// Canale 6 - Totale pacchi quinto codice - parziale
Counters[6].Enable := TRUE;
Counters[6].Nome := CONCAT(STR1:= 'Quinto codice - parziale, VALORE -> ', STR2 := INT_TO_STRING(5));
Counters[6].Enable_Reset_Storico := FALSE;
Counters[6].ResetCounter := DATA_LOGGER.Reset_Operatore;
Counters[6].Daily_Reference_Total := Counters[1].Daily_Counter_State;
Counters[6].Weekly_Reference_Total := Counters[1].Weekly_Counter_State;
Counters[6].Periodic_Reference_Total := TotalePacchiParziali;
Counters[6].Enable_Reset_Dopo_Salvataggio := TRUE;

// Canale 7 - Totale pacchi sesto codice - parziale
Counters[7].Enable := TRUE;
Counters[7].Nome := CONCAT(STR1:= 'Sesto codice - parziale, VALORE -> ', STR2 := INT_TO_STRING(6));
Counters[7].Enable_Reset_Storico := FALSE;
Counters[7].ResetCounter := DATA_LOGGER.Reset_Operatore;
Counters[7].Daily_Reference_Total := Counters[1].Daily_Counter_State;
Counters[7].Weekly_Reference_Total := Counters[1].Weekly_Counter_State;
Counters[7].Periodic_Reference_Total := TotalePacchiParziali;
Counters[7].Enable_Reset_Dopo_Salvataggio := TRUE;

// Canale 8 - Totale pacchi settimo codice - parziale
Counters[8].Enable := TRUE;
Counters[8].Nome := CONCAT(STR1:= 'Settimo codice - parziale, VALORE -> ', STR2 := INT_TO_STRING(7));
Counters[8].Enable_Reset_Storico := FALSE;
Counters[8].ResetCounter := DATA_LOGGER.Reset_Operatore;
Counters[8].Daily_Reference_Total := Counters[1].Daily_Counter_State;
Counters[8].Weekly_Reference_Total := Counters[1].Weekly_Counter_State;
Counters[8].Periodic_Reference_Total := TotalePacchiParziali;
Counters[8].Enable_Reset_Dopo_Salvataggio := TRUE;

// Canale 9 - Totale pacchi ottavo codice - parziale
Counters[9].Enable := TRUE;
Counters[9].Nome := CONCAT(STR1:= 'Ottavo codice - parziale, VALORE -> ', STR2 := INT_TO_STRING(8));
Counters[9].Enable_Reset_Storico := FALSE;
Counters[9].ResetCounter := DATA_LOGGER.Reset_Operatore;
Counters[9].Daily_Reference_Total := Counters[1].Daily_Counter_State;
Counters[9].Weekly_Reference_Total := Counters[1].Weekly_Counter_State;
Counters[9].Periodic_Reference_Total := TotalePacchiParziali;
Counters[9].Enable_Reset_Dopo_Salvataggio := TRUE;

// Canale 10 - Totale pacchi nono codice - parziale
Counters[10].Enable := TRUE;
Counters[10].Nome := CONCAT(STR1:= 'Nono codice - parziale, VALORE -> ', STR2 := INT_TO_STRING(9));
Counters[10].Enable_Reset_Storico := FALSE;
Counters[10].ResetCounter := DATA_LOGGER.Reset_Operatore;
Counters[10].Daily_Reference_Total := Counters[1].Daily_Counter_State;
Counters[10].Weekly_Reference_Total := Counters[1].Weekly_Counter_State;
Counters[10].Periodic_Reference_Total := TotalePacchiParziali;
Counters[10].Enable_Reset_Dopo_Salvataggio := TRUE;

// Canale 11 - Totale pacchi decimo codice - parziale
Counters[11].Enable := TRUE;
Counters[11].Nome := CONCAT(STR1:= 'Decimo codice - parziale, VALORE -> ', STR2 := INT_TO_STRING(10));
Counters[11].Enable_Reset_Storico := FALSE;
Counters[11].ResetCounter := DATA_LOGGER.Reset_Operatore;
Counters[11].Daily_Reference_Total := Counters[1].Daily_Counter_State;
Counters[11].Weekly_Reference_Total := Counters[1].Weekly_Counter_State;
Counters[11].Periodic_Reference_Total := TotalePacchiParziali;
Counters[11].Enable_Reset_Dopo_Salvataggio := TRUE;

// Canale 12 - Totale pacchi undicesimo codice - parziale
Counters[12].Enable := TRUE;
Counters[12].Nome := CONCAT(STR1:= 'Undicesimo codice - parziale, VALORE -> ', STR2 := INT_TO_STRING(11));
Counters[12].Enable_Reset_Storico := FALSE;
Counters[12].ResetCounter := DATA_LOGGER.Reset_Operatore;
Counters[12].Daily_Reference_Total := Counters[1].Daily_Counter_State;
Counters[12].Weekly_Reference_Total := Counters[1].Weekly_Counter_State;
Counters[12].Periodic_Reference_Total := TotalePacchiParziali;
Counters[12].Enable_Reset_Dopo_Salvataggio := TRUE;

// Canale 13 - Totale pacchi dodicesimo codice - parziale
Counters[13].Enable := TRUE;
Counters[13].Nome := CONCAT(STR1:= 'Dodicesimo codice - parziale, VALORE -> ', STR2 := INT_TO_STRING(12));
Counters[13].Enable_Reset_Storico := FALSE;
Counters[13].ResetCounter := DATA_LOGGER.Reset_Operatore;
Counters[13].Daily_Reference_Total := Counters[1].Daily_Counter_State;
Counters[13].Weekly_Reference_Total := Counters[1].Weekly_Counter_State;
Counters[13].Periodic_Reference_Total := TotalePacchiParziali;
Counters[13].Enable_Reset_Dopo_Salvataggio := TRUE;

// Canale 14 - Totale pacchi tredicesimo codice - parziale
Counters[14].Enable := TRUE;
Counters[14].Nome := CONCAT(STR1:= 'Tredicesimo codice - parziale, VALORE -> ', STR2 := INT_TO_STRING(13));
Counters[14].Enable_Reset_Storico := FALSE;
Counters[14].ResetCounter := DATA_LOGGER.Reset_Operatore;
Counters[14].Daily_Reference_Total := Counters[1].Daily_Counter_State;
Counters[14].Weekly_Reference_Total := Counters[1].Weekly_Counter_State;
Counters[14].Periodic_Reference_Total := TotalePacchiParziali;
Counters[14].Enable_Reset_Dopo_Salvataggio := TRUE;

// Canale 15 - Totale pacchi quattordicesimo codice - parziale
Counters[15].Enable := TRUE;
Counters[15].Nome := CONCAT(STR1:= 'Quattordicesimo codice - parziale, VALORE -> ', STR2 := INT_TO_STRING(14));
Counters[15].Enable_Reset_Storico := FALSE;
Counters[15].ResetCounter := DATA_LOGGER.Reset_Operatore;
Counters[15].Daily_Reference_Total := Counters[1].Daily_Counter_State;
Counters[15].Weekly_Reference_Total := Counters[1].Weekly_Counter_State;
Counters[15].Periodic_Reference_Total := TotalePacchiParziali;
Counters[15].Enable_Reset_Dopo_Salvataggio := TRUE;

// Canale 16 - Totale pacchi quindicesimo codice - parziale
Counters[16].Enable := TRUE;
Counters[16].Nome := CONCAT(STR1:= 'Quindicesimo codice - parziale, VALORE -> ', STR2 := INT_TO_STRING(15));
Counters[16].Enable_Reset_Storico := FALSE;
Counters[16].ResetCounter := DATA_LOGGER.Reset_Operatore;
Counters[16].Daily_Reference_Total := Counters[1].Daily_Counter_State;
Counters[16].Weekly_Reference_Total := Counters[1].Weekly_Counter_State;
Counters[16].Periodic_Reference_Total := TotalePacchiParziali;
Counters[16].Enable_Reset_Dopo_Salvataggio := TRUE;

(* Reset x evitare false letture *)
PaccoPresoXDataLogger := FALSE;
//DATA_LOGGER.Reset_Operatore := FALSE;
END_ACTION

ACTION _09_CalcolaFormatura:
//Ack 
IF HMI_ErrAckCalcolaFormatura THEN
	HMI_Forming_ErroreCalcoli := 0;
	HMI_ErrAckCalcolaFormatura := FALSE;
	FOR i:= 1 TO MAXFORMING DO
		HMI_Forming_FormaturaAttivata[i] := FALSE;
	END_FOR
END_IF

//Attivazione
FOR i:= 1 TO MAXFORMING DO
	//IF HMI_Forming_Attivazione[i] AND i <=2 AND FALSE THEN
	IF HMI_Forming_Attivazione[i] AND i <=3 AND FALSE THEN
		NCodiciPresenti := 0;
		FOR iform := 1 TO MAXFORMING DO
			FOR icode:=1 TO MAXFORMINGCODE DO
				FOR icode2:=1 TO MAXFORMINGCODE DO
					IF HMI_Forming_CodiciAbilitatiFormatura[i].Code[icode] = Forming[iform].Code[icode] AND Forming[iform].Code[icode] > 0 AND iform <> i THEN
						HMI_Forming_ErroreCalcoli := ErrRipetizioneCodici;		
						HMI_Forming_Attivazione[i] := FALSE; // prueva quitar 
						RETURN;
					END_IF 
				END_FOR
				IF HMI_Forming_CodiciAbilitatiFormatura[i].Code[icode] > 0 THEN
					NCodiciPresenti := NcodiciPresenti+1;
				END_IF
			END_FOR
		END_FOR
		//VErifico che ci sia almento un codice da attivare
		IF NcodiciPresenti = 0 THEN
			HMI_Forming_ErroreCalcoli := ErrNessunCodiciPresente;
			RETURN;
		END_IF
	
		// MEMSET(ADR(Forming[i]),0,SIZEOF(Forming[i])); //prueva Quitar
		IF NOT CalcolaFormaturaTrig AND FALSE  THEN
			HMI_Forming_FormaturaAttivata[i] 	:= FALSE;
			TFCalcoloFormatura.PulisciMemoria 	:= TRUE;
			IF TFCalcoloFormatura.PulisciMemoriaDone THEN	
				HMI_Forming_ErroreCalcoli := 0;
				//Assegno l'ordine tutto a 1 perchè ho solo lastre
				FOR i:= 1 TO MAXFORMINGSLAB DO
					IF i <= HMI_Forming_NumeroElementiDaDepositare THEN
						TFCalcoloFormatura.TipoElementoDep[i] := LASTRA;//Settiamo tutte lastre!!
					ELSE
						TFCalcoloFormatura.TipoElementoDep[i] := TERMINATORE;//Settiamo il resto come terminatore
					END_IF
				END_FOR
				TFCalcoloFormatura.Materiale[e_Tipo_Elemento_Da_Lavorare.LASTRA]		:= HMI_Forming_LastraDaDepositare;
				TFCalcoloFormatura.Materiale[e_Tipo_Elemento_Da_Lavorare.LASTRA].Typology := LASTRA;
				TFCalcoloFormatura.Materiale[e_Tipo_Elemento_Da_Lavorare.FALDA]			:= HMI_Forming_LastraDaDepositare;
				TFCalcoloFormatura.Materiale[e_Tipo_Elemento_Da_Lavorare.FALDA].Typology := FALDA;
				TFCalcoloFormatura.Materiale[e_Tipo_Elemento_Da_Lavorare.QUADROTTA]		:= HMI_Forming_LastraDaDepositare;
				TFCalcoloFormatura.Materiale[e_Tipo_Elemento_Da_Lavorare.QUADROTTA].Typology := QUADROTTA;
				TFCalcoloFormatura.Supporto			:= HMI_Forming_Supporto;	//Assegno la tipologia di supporto
				TFCalcoloFormatura.CalcolaFormatura := TRUE; 		//Lancio esecuzione dei calcoli
				MEMSET(ADR(HMI_Forming_FormaturaCalcolata),0,SIZEOF(HMI_Forming_FormaturaCalcolata));	//Pulisco la memoria di destinazione
				CalcolaFormaturaTrig := TRUE;
				HMI_Forming_Attivazione[i] := FALSE;
				TFCalcoloFormatura.PulisciMemoria := FALSE;
			END_IF
		ELSIF (TFCalcoloFormatura.CalcolaFormaturaDone OR TFCalcoloFormatura.Errore > 0) AND CalcolaFormaturaTrig AND FALSE THEN
			TFCalcoloFormatura.CalcolaFormatura := FALSE;
			IF TFCalcoloFormatura.Errore = 0 THEN
				IDFormatura 			:= IDFormatura+1;
				GUIDFormatura 			:= STRING_TO_UINT(concat(UINT_TO_STRING(NUMERO_MACCHINA),UINT_TO_STRING(IDFormatura)));
				HMI_Forming_GUID 		:= GUIDFormatura;
		
				HMI_Forming_FormaturaCalcolata 	:= TFCalcoloFormatura.FormingSlab;
				MEMSET(ADR(Forming[i]),0,SIZEOF(Forming[i]));	//Pulisco la memoria di destinazione
				Forming[i] 							:= TFCalcoloFormatura.FormingSlab;
				Forming[i].Enable 					:= 1;
				Forming[i].Code 					:= HMI_Forming_CodiciAbilitatiFormatura[i].Code;
				Forming[i].GUID						:= HMI_Forming_GUID;
				Forming[i].Pallet					:= HMI_Forming_Supporto;
				HMI_Forming_IndiceFormaturaAttivata := i;
				HMI_Forming_FormaturaAttivata[i] 	:= TRUE;
			ELSE
				HMI_Forming_ErroreCalcoli := TFCalcoloFormatura.Errore;
			END_IF
			CalcolaFormaturaTrig := FALSE;
			HMI_Forming_Attivazione[i] := FALSE;
		END_IF
	ELSIF HMI_Forming_Attivazione[i] AND FALSE THEN
		memset(destAddr:=ADR(TFCalcoloFormatura.Errore),fillByte:=(UINT_TO_USINT(ErrNumeroMassimoFormatureAmmesse)),n:=SIZEOF(TFCalcoloFormatura.Errore));
	END_IF

	//Disattivazione formatura
	IF HMI_Forming_Disattivazione[i] AND FALSE  THEN
		HMI_Forming_Disattivazione[i] := FALSE;
		MEMSET(ADR(Forming[i]),0,SIZEOF(Forming[i]));	//Pulisco la formatura selezionata e di consegenza la disattivo
	END_IF
		
END_FOR

//IF HMI_Forming_Calcola AND Forming[1].Enable = 1 AND Forming[2].Enable = 1 THEN
//	memset(destAddr:=ADR(TFCalcoloFormatura.Errore),fillByte:=(UINT_TO_USINT(ErrNumeroMassimoFormatureAmmesse)),n:=SIZEOF(TFCalcoloFormatura.Errore));
//	HMI_Forming_Calcola := FALSE;
//Creazione
IF HMI_Forming_Calcola  AND NOT CalcolaFormaturaTrig AND FALSE THEN
	TFCalcoloFormatura.PulisciMemoria := TRUE;
	IF TFCalcoloFormatura.PulisciMemoriaDone THEN	
		HMI_Forming_ErroreCalcoli := 0;
		//Assegno l'ordine tutto a 1 perchè ho solo lastre
		FOR i:= 1 TO MAXFORMINGSLAB DO
			IF i <= HMI_Forming_NumeroElementiDaDepositare THEN
				TFCalcoloFormatura.TipoElementoDep[i] := LASTRA;//Settiamo tutte lastre!!
			ELSE
				TFCalcoloFormatura.TipoElementoDep[i] := TERMINATORE;//Settiamo il resto come terminatore
			END_IF
		END_FOR
		TFCalcoloFormatura.Materiale[e_Tipo_Elemento_Da_Lavorare.LASTRA]		:= HMI_Forming_LastraDaDepositare;
		TFCalcoloFormatura.Materiale[e_Tipo_Elemento_Da_Lavorare.LASTRA].Typology := LASTRA;
		TFCalcoloFormatura.Materiale[e_Tipo_Elemento_Da_Lavorare.FALDA]			:= HMI_Forming_LastraDaDepositare;
		TFCalcoloFormatura.Materiale[e_Tipo_Elemento_Da_Lavorare.FALDA].Typology := FALDA;
		TFCalcoloFormatura.Materiale[e_Tipo_Elemento_Da_Lavorare.QUADROTTA]		:= HMI_Forming_LastraDaDepositare;
		TFCalcoloFormatura.Materiale[e_Tipo_Elemento_Da_Lavorare.QUADROTTA].Typology := QUADROTTA;
		TFCalcoloFormatura.Supporto					:= HMI_Forming_Supporto;	//Assegno la tipologia di supporto
		TFCalcoloFormatura.CalcolaFormatura 		:= HMI_Forming_Calcola; 		//Lancio esecuzione dei calcoli
		TFCalcoloFormatura.NumeroElementiDaDepositare := HMI_Forming_NumeroElementiDaDepositare; 		//Lancio esecuzione dei calcoli
			
		MEMSET(ADR(HMI_Forming_FormaturaCalcolata),0,SIZEOF(HMI_Forming_FormaturaCalcolata));	//Pulisco la memoria di destinazione
		CalcolaFormaturaTrig := TRUE;
		//HMI_Forming_Calcola := FALSE;
		TFCalcoloFormatura.PulisciMemoria := FALSE;
	END_IF

ELSIF HMI_Forming_Calcola AND (TFCalcoloFormatura.CalcolaFormaturaDone OR TFCalcoloFormatura.Errore > 0) AND CalcolaFormaturaTrig AND FALSE THEN
	HMI_Forming_Calcola := FALSE;
	TFCalcoloFormatura.CalcolaFormatura := FALSE;
	IF TFCalcoloFormatura.Errore = 0 THEN
		HMI_Forming_FormaturaCalcolata 	:= TFCalcoloFormatura.FormingSlab;
	//	IDFormatura 			:= IDFormatura+1;
	//	GUIDFormatura 			:= STRING_TO_UINT(concat(UINT_TO_STRING(NUMERO_MACCHINA),UINT_TO_STRING(IDFormatura)));
	//	HMI_Forming_GUID 		:= GUIDFormatura;
		(*FOR i:= 1 TO 2 DO
			IF Forming[i].Enable <> 1 THEN
				MEMSET(ADR(Forming[i]),0,SIZEOF(Forming[i]));	//Pulisco la memoria di destinazione
				HMI_Forming_IndiceFormaturaAttivata := i;
				Forming[i] 			:= TFCalcoloFormatura.FormingSlab;
				Forming[i].Enable 	:= 1;
				Forming[i].Code 	:= HMI_Forming_CodiciAbilitatiFormatura[i].Code;
				Forming[i].GUID		:= HMI_Forming_GUID;
				Forming[i].Pallet	:= HMI_Forming_Supporto;
			ELSE
				CONTINUE;
			END_IF
			EXIT;
		END_FOR*)
		HMI_Forming_FormaturaCreata := TRUE;
	ELSE
		HMI_Forming_ErroreCalcoli := TFCalcoloFormatura.Errore;
	END_IF
	
	CalcolaFormaturaTrig := FALSE;
END_IF
IF FALSE THEN 
	 TFCalcoloFormatura();
END_IF
  

(*//Ack 
IF HMI_ErrAckCalcolaFormatura THEN
	HMI_Forming_ErroreCalcoli := 0;
	HMI_ErrAckCalcolaFormatura := FALSE;
	FOR i:= 1 TO MAXFORMING DO
		HMI_ConfermaAttivazioneFormatura[i] := FALSE;
		HMI_Forming_FormaturaAttivata[i] := FALSE;
	END_FOR
END_IF

//Attivazione
FOR i:= 1 TO MAXFORMING DO
	IF HMI_Forming_Attivazione[i] AND i <=2 THEN
		NCodiciPresenti := 0;
		
		FOR iform := 1 TO MAXFORMING DO
			FOR icode:=1 TO MAXFORMINGCODE DO
				FOR icode2:=1 TO MAXFORMINGCODE DO
					IF HMI_Forming_CodiciAbilitatiFormatura[i].Code[icode] = Forming[iform].Code[icode] AND Forming[iform].Code[icode] > 0 AND iform <> i THEN
						HMI_Forming_ErroreCalcoli := ErrRipetizioneCodici;		
						HMI_Forming_Attivazione[i] := FALSE;
						RETURN;
					END_IF 
				END_FOR
				IF HMI_Forming_CodiciAbilitatiFormatura[i].Code[icode] > 0 THEN
					NCodiciPresenti := NcodiciPresenti+1;
				END_IF
			END_FOR
		END_FOR
		//VErifico che ci sia almento un codice da attivare
		IF NcodiciPresenti = 0 THEN
			HMI_Forming_ErroreCalcoli := ErrNessunCodiciPresente;
			RETURN;
		END_IF
	
		MEMSET(ADR(Forming[i]),0,SIZEOF(Forming[i]));
		IF NOT CalcolaFormaturaTrig  THEN
			HMI_Forming_FormaturaAttivata[i] 	:= FALSE;
			TFCalcoloFormatura.PulisciMemoria 	:= TRUE;
			IF TFCalcoloFormatura.PulisciMemoriaDone THEN	
				HMI_Forming_ErroreCalcoli := 0;
				//Assegno l'ordine tutto a 1 perchè ho solo lastre
				FOR i:= 1 TO MAXFORMINGSLAB DO
					IF i <= HMI_Forming_NumeroElementiDaDepositare THEN
						TFCalcoloFormatura.TipoElementoDep[i] := LASTRA;//Settiamo tutte lastre!!
					ELSE
						TFCalcoloFormatura.TipoElementoDep[i] := TERMINATORE;//Settiamo il resto come terminatore
					END_IF
				END_FOR
				TFCalcoloFormatura.Materiale[e_Tipo_Elemento_Da_Lavorare.LASTRA]		:= HMI_Forming_LastraDaDepositare;
				TFCalcoloFormatura.Materiale[e_Tipo_Elemento_Da_Lavorare.LASTRA].Typology := LASTRA;
				TFCalcoloFormatura.Materiale[e_Tipo_Elemento_Da_Lavorare.FALDA]			:= HMI_Forming_LastraDaDepositare;
				TFCalcoloFormatura.Materiale[e_Tipo_Elemento_Da_Lavorare.FALDA].Typology := FALDA;
				TFCalcoloFormatura.Materiale[e_Tipo_Elemento_Da_Lavorare.QUADROTTA]		:= HMI_Forming_LastraDaDepositare;
				TFCalcoloFormatura.Materiale[e_Tipo_Elemento_Da_Lavorare.QUADROTTA].Typology := QUADROTTA;
				TFCalcoloFormatura.Supporto			:= HMI_Forming_Supporto;	//Assegno la tipologia di supporto
				TFCalcoloFormatura.CalcolaFormatura := TRUE; 		//Lancio esecuzione dei calcoli
				MEMSET(ADR(HMI_Forming_FormaturaCalcolata),0,SIZEOF(HMI_Forming_FormaturaCalcolata));	//Pulisco la memoria di destinazione
				HMI_Forming_Attivazione[i] := FALSE;
				TFCalcoloFormatura.PulisciMemoria := FALSE;
				CalcolaFormaturaTrig := TRUE;
			END_IF
		ELSIF (TFCalcoloFormatura.CalcolaFormaturaDone OR TFCalcoloFormatura.Errore > 0) AND CalcolaFormaturaTrig THEN
			//CalcolaFormaturaTrig := FALSE;
			TFCalcoloFormatura.CalcolaFormatura := FALSE;
			IF TFCalcoloFormatura.Errore = 0 THEN
				IDFormatura 			:= IDFormatura+1;
				GUIDFormatura 			:= STRING_TO_UINT(concat(UINT_TO_STRING(NUMERO_MACCHINA),UINT_TO_STRING(IDFormatura)));
				HMI_Forming_GUID 		:= GUIDFormatura;
		
				HMI_Forming_FormaturaCalcolata 	:= TFCalcoloFormatura.FormingSlab;
				MEMSET(ADR(Forming[i]),0,SIZEOF(Forming[i]));	//Pulisco la memoria di destinazione
				Forming[i] 							:= TFCalcoloFormatura.FormingSlab;
				Forming[i].Enable 					:= 1;
				Forming[i].Code 					:= HMI_Forming_CodiciAbilitatiFormatura[i].Code;
				Forming[i].GUID						:= HMI_Forming_GUID;
				Forming[i].Pallet					:= HMI_Forming_Supporto;
				HMI_Forming_IndiceFormaturaAttivata := i;
				HMI_Forming_FormaturaAttivata[i] 	:= TRUE;
			ELSE
				HMI_Forming_ErroreCalcoli := TFCalcoloFormatura.Errore;
			END_IF
			HMI_Forming_Attivazione[i] := FALSE;
		END_IF
	ELSIF HMI_Forming_Attivazione[i] THEN
		memset(destAddr:=ADR(TFCalcoloFormatura.Errore),fillByte:=(UINT_TO_USINT(ErrNumeroMassimoFormatureAmmesse)),n:=SIZEOF(TFCalcoloFormatura.Errore));
	END_IF

	//Disattivazione formatura
	IF HMI_Forming_Disattivazione[i] THEN
		HMI_Forming_Disattivazione[i] := FALSE;
		MEMSET(ADR(Forming[i]),0,SIZEOF(Forming[i]));	//Pulisco la formatura selezionata e di consegenza la disattivo
	END_IF
		
END_FOR

//IF HMI_Forming_Calcola AND Forming[1].Enable = 1 AND Forming[2].Enable = 1 THEN
//	memset(destAddr:=ADR(TFCalcoloFormatura.Errore),fillByte:=(UINT_TO_USINT(ErrNumeroMassimoFormatureAmmesse)),n:=SIZEOF(TFCalcoloFormatura.Errore));
//	HMI_Forming_Calcola := FALSE;
//Creazione
IF HMI_Forming_Calcola  AND NOT CalcolaFormaturaTrig  THEN
	TFCalcoloFormatura.PulisciMemoria := TRUE;
	IF TFCalcoloFormatura.PulisciMemoriaDone THEN	
		TFCalcoloFormatura.PulisciMemoria := FALSE;
		HMI_Forming_ErroreCalcoli := 0;
		CalcolaFormaturaTrig := TRUE;
		//Assegno l'ordine tutto a 1 perchè ho solo lastre
		FOR i:= 1 TO MAXFORMINGSLAB DO
			IF i <= HMI_Forming_NumeroElementiDaDepositare THEN
				TFCalcoloFormatura.TipoElementoDep[i] := LASTRA;//Settiamo tutte lastre!!
			ELSE
				TFCalcoloFormatura.TipoElementoDep[i] := TERMINATORE;//Settiamo il resto come terminatore
			END_IF
		END_FOR
		TFCalcoloFormatura.Materiale[e_Tipo_Elemento_Da_Lavorare.LASTRA]		:= HMI_Forming_LastraDaDepositare;
		TFCalcoloFormatura.Materiale[e_Tipo_Elemento_Da_Lavorare.LASTRA].Typology := LASTRA;
		TFCalcoloFormatura.Materiale[e_Tipo_Elemento_Da_Lavorare.FALDA]			:= HMI_Forming_LastraDaDepositare;
		TFCalcoloFormatura.Materiale[e_Tipo_Elemento_Da_Lavorare.FALDA].Typology := FALDA;
		TFCalcoloFormatura.Materiale[e_Tipo_Elemento_Da_Lavorare.QUADROTTA]		:= HMI_Forming_LastraDaDepositare;
		TFCalcoloFormatura.Materiale[e_Tipo_Elemento_Da_Lavorare.QUADROTTA].Typology := QUADROTTA;
		TFCalcoloFormatura.Supporto					:= HMI_Forming_Supporto;	//Assegno la tipologia di supporto
		TFCalcoloFormatura.CalcolaFormatura 		:= HMI_Forming_Calcola; 		//Lancio esecuzione dei calcoli
		TFCalcoloFormatura.NumeroElementiDaDepositare := HMI_Forming_NumeroElementiDaDepositare; 		//Lancio esecuzione dei calcoli
			
		MEMSET(ADR(HMI_Forming_FormaturaCalcolata),0,SIZEOF(HMI_Forming_FormaturaCalcolata));	//Pulisco la memoria di destinazione
		//HMI_Forming_Calcola := FALSE;
	END_IF

ELSIF HMI_Forming_Calcola AND (TFCalcoloFormatura.CalcolaFormaturaDone OR TFCalcoloFormatura.Errore > 0) AND CalcolaFormaturaTrig THEN
	HMI_Forming_Calcola := FALSE;
	TFCalcoloFormatura.CalcolaFormatura := FALSE;
	IF TFCalcoloFormatura.Errore = 0 THEN
		HMI_Forming_FormaturaCalcolata 	:= TFCalcoloFormatura.FormingSlab;
	//	IDFormatura 			:= IDFormatura+1;
	//	GUIDFormatura 			:= STRING_TO_UINT(concat(UINT_TO_STRING(NUMERO_MACCHINA),UINT_TO_STRING(IDFormatura)));
	//	HMI_Forming_GUID 		:= GUIDFormatura;
		(*FOR i:= 1 TO 2 DO
			IF Forming[i].Enable <> 1 THEN
				MEMSET(ADR(Forming[i]),0,SIZEOF(Forming[i]));	//Pulisco la memoria di destinazione
				HMI_Forming_IndiceFormaturaAttivata := i;
				Forming[i] 			:= TFCalcoloFormatura.FormingSlab;
				Forming[i].Enable 	:= 1;
				Forming[i].Code 	:= HMI_Forming_CodiciAbilitatiFormatura[i].Code;
				Forming[i].GUID		:= HMI_Forming_GUID;
				Forming[i].Pallet	:= HMI_Forming_Supporto;
			ELSE
				CONTINUE;
			END_IF
			EXIT;
		END_FOR*)
		HMI_Forming_FormaturaCreata := TRUE;
	ELSE
		HMI_Forming_ErroreCalcoli := TFCalcoloFormatura.Errore;
	END_IF
	
	CalcolaFormaturaTrig := FALSE;
END_IF

TFCalcoloFormatura();*)
END_ACTION

ACTION _10_PackModifier:
//Filtro le FTC delle postazioni
FOR i := 1 TO MAXAREAPRESENT DO
	FiltroFTCPalletPerManuale[i].FilterTime_OFF := 3000;
	FiltroFTCPalletPerManuale[i].FilterTime_ON 	:= 3000;
	FiltroFTCPalletPerManuale[i].IN_Signal 		:= I_PHPresenzaPallet[i];
	FiltroFTCPalletPerManuale[i]();
END_FOR

IF MachinePalletizer_TF.CmdExe.Code = CmdNOP THEN
	FOR i:= 1 TO MAXAREAPRESENT DO
		IF HMI_NumeroPezziPresentiPostazione[i] <> WorkAreaState[i].P-1 THEN
			WorkAreaState[i].P := HMI_NumeroPezziPresentiPostazione[i]+1;
		END_IF	
		
		IF HMI_NumeroPezziPresentiCavallete[i].HMI_NumeroPezziPresentiPostazione_A_Cavaleto <> WorkAreaState[i].P_Cava.HMI_NumeroPezziPresentiPostazione_A_Cavaleto -1	THEN 
			WorkAreaState[i].P_Cava.HMI_NumeroPezziPresentiPostazione_A_Cavaleto 
								:= HMI_NumeroPezziPresentiCavallete[i].HMI_NumeroPezziPresentiPostazione_A_Cavaleto +1 ;
		END_IF
		IF HMI_NumeroPezziPresentiCavallete[i].HMI_NumeroPezziPresentiPostazione_B_Cavaleto <> WorkAreaState[i].P_Cava.HMI_NumeroPezziPresentiPostazione_B_Cavaleto -1	THEN 
			WorkAreaState[i].P_Cava.HMI_NumeroPezziPresentiPostazione_B_Cavaleto 
								:= HMI_NumeroPezziPresentiCavallete[i].HMI_NumeroPezziPresentiPostazione_B_Cavaleto +1 ;
		END_IF
		IF (ActualPickingListFromHMI[1].State <> 0 OR ActualPickingListFromHMI[2].State <> 0 OR ActualPickingListFromHMI[3].State <>0)
				AND WorkAreaState[i].Supporto.Tipologia = CAVALLETTO THEN 
			WorkAreaState[i].P := HMI_NumeroPezziPresentiCavallete[i].HMI_NumeroPezziPresentiPostazione_A_Cavaleto 
					+ HMI_NumeroPezziPresentiCavallete[i].HMI_NumeroPezziPresentiPostazione_B_Cavaleto +1 ;
		END_IF		
		
		IF WorkAreaState[i].PackPointerModified THEN//Se sto facendo una modifica da HMI
			WorkAreaState[i].PackPointer:= MIN(MAX(1,WorkAreaState[i].PackPointer ),MAXFORMINGSLAB);//limito i valori con quelli ammissibili
			IF WorkAreaState[i].PackPointer > WorkAreaState[i].P THEN 
				IF (WorkAreaState[i].PackPointer - WorkAreaState[i].P) = 1 THEN
					WorkAreaState[i].P := WorkAreaState[i].P+1;
				ELSE 
					WorkAreaState[i].P := WorkAreaState[i].PackPointer+1;	
				END_IF
			ELSE
				IF (WorkAreaState[i].PackPointer - WorkAreaState[i].P) = -1 THEN
					WorkAreaState[i].P := WorkAreaState[i].P-1;
				ELSE 
					WorkAreaState[i].P := WorkAreaState[i].PackPointer+1;	
				END_IF
			END_IF
			WorkAreaState[i].Slow := 1;
			WorkAreaState[i].PackPointerModified := FALSE;
			WorkAreaState[i].PackPointer := -1;
		END_IF
		//
		HMI_NumeroPezziPresentiPostazione[i] := MAX(0,WorkAreaState[i].P-1);
		
		AggiuntaPalletManuale(WorkArea := ADR(WorkArea),
									WorkAreaState := ADR(WorkAreaState),
									WorkAreaNumber := i,
									Forming := ADR(Forming),
									Pallet := ADR(Pallet),
									Layer := ADR(Layer),
									ProgressiveNrWA := ADR(ProgressiveNrWA),
									CodicePostazione := WorkAreaState[i].Code,
									AbilitaAssegnazioneCodicePiazzoleConPaccoSuRibaltino := TRUE,
									PH_Presenza := FiltroFTCPalletPerManuale[i].Out_Signal_Filtrato);	
	END_FOR
END_IF
END_ACTION

ACTION _11_CalcolaListaProduzione:
{region "Gestione zona GLOBALE - Postazioni da 1 a 8"}


//#############################################################################################################

{region "Gestione zona GLOBALE - Postazioni da 1 a 8"}

//Traferisco i valori dei supporti della lista 1 nella lista 2 e 3
 

FOR LoopLista := 1 TO 3 DO
	IdxLista := LoopLista;		 
	 // IdxLista := 2;		  
	CASE IdxLista OF	 
		1: Iforstart := 1; Iforend := MAXAREAPRESENT;
		2: Iforstart := 1; Iforend := 4;
		3: Iforstart := 5; Iforend := MAXAREAPRESENT;
	END_CASE	 
	IF MachinePalletizer_TF.IN.Mode.Man AND
		(MachinePalletizer_TF.CmdExe.Code = CmdNOP OR MachinePalletizer_TF.CmdExe.Code = CmdMAN) THEN

//--------------------------------------------------------
			//AZZERAMENTO (Reset) lista di picking	
//--------------------------------------------------------		 
			IF Cmd_AzzeraLista[IdxLista] THEN
				IF Prueva THEN
					MissionClr := ADR(Mission) ;
	 				MEMSET(destAddr := ADR(MissionClr^),fillByte := 0 , n := SIZEOF(MissionClr^));
				END_IF
					ClrEstructura := ADR(PosCavalleteOrdenPikin) ;
					MEMSET(destAddr := ADR(ClrEstructura^),fillByte := 0 , n := SIZEOF(ClrEstructura^));	  
					NuEstacionesPiking := 0 ;	  
					NuEstacionPiking   := 0 ;
					NuPosGuiroPiking := 0;
					PosFinOrdenPikingCaballete := 0 ;
					
					MultiplesCavalletesReceta := FALSE ;
					CoordenadaPasillo0_Y := 0 ;
					CoordenadaPasillo180_Y := 0 ;
				
				//FOR i:= 1 TO 3 DO
						//CalcolaFormingRT2[i] := FALSE ;
					CalcolaFormingRT[IdxLista] := FALSE ;
					CalcolaFormingRT2[IdxLista] := FALSE ;	 
						//#Añadido 4_7_2025########################
					Formacion_bandelCalOk[IdxLista]			:= FALSE ;
					Formacion_FrameCalOk[IdxLista]			:= FALSE ;
					Formacion_De_listaOk[IdxLista]			:= FALSE ;
					FormaturaAFRAMERT[IdxLista]		   	:=	FormingEmpty;
					FormaturaBundleRT[IdxLista]	 		:=	FormingEmpty;
					
					MEMSET(destAddr := ADR(TFFormacionBandelCalculada),fillByte := 0 , n := SIZEOF(TFFormacionBandelCalculada));
					MEMSET(destAddr := ADR(TFFormacionCavalleteCalculada),fillByte := 0 , n := SIZEOF(TFFormacionCavalleteCalculada));
					MEMSET(destAddr := ADR(TFCalcoloFormaturaWA),fillByte := 0 , n := SIZEOF(TFCalcoloFormaturaWA));
					MEMSET(destAddr := ADR(GestionCargaCaballete),fillByte := 0 , n := SIZEOF(GestionCargaCaballete));	
					MEMSET(destAddr := ADR(GestionDescargaCaballete),fillByte := 0 , n := SIZEOF(GestionDescargaCaballete));			  
				//Añadido 4_7_2025##########################
						
				// END_FOR
				ActualPickingListFromHMI[IdxLista].State := e_StatoWorkOrder.NON_ESEGUITO;
				HMI_NumeroLastreDepOrdineAttuale[IdxLista] := 0; 
				//Disattivazione formatura
				Forming[1] := FormingEmpty;	//Pulisco la formatura selezionata e di consegenza la disattivo
				Forming[2] := FormingEmpty;	//Pulisco la formatura selezionata e di consegenza la disattivo
				Forming[3] := FormingEmpty;	//Pulisco la formatura selezionata e di consegenza la disattivo
				Forming[4] := FormingEmpty;	//Pulisco la formatura selezionata e di consegenza la disattivo
				ActualPickingListFromHMI[IdxLista].State := e_StatoWorkOrder.NON_ESEGUITO;
				Cmd_AttivaLista[IdxLista] := FALSE;
				HMI_Forming_NumeroElementiDaDepositare := 0;
 				RequestPickingListFromHMI[IdxLista].SlabNumber :=0;
	 
				//Azzero le liste per le postazioni dove non avviene la pallettizzazione
				FOR i:= Iforstart TO Iforend DO	
					TFClearWorkAreaArray(ADR(Workarea),ADR(WorkAreaState),k:=i);
					HMI_WorkAreaDataPicking[i].Destinazione := FALSE;
					HMI_WorkAreaDataPicking[i].NumElementiDaLavorare := 0;
					WorkAreaState[i].P 			:= 1;
					WorkAreaProductionList[i] 	:= ListaEmpty;
					WorkAreaOffset[i].Y 		:= 0;
					//HMI_NumeroPezziPresentiPostazione[i] 	:= 0; // Quitado Para No resetear posiciones
					NumeroPezziPresentiPostazioneStart[i] 	:= 0;
					WorkAreaProductionList[i].Stato 		:= e_Stato_ListaDiProduzione.LISTA_PROD_ASSENTE;	 
				END_FOR			  
				ActualPickingListFromHMI[IdxLista].SlabNumber 		  			:= 0;
				ActualPickingListFromHMI[IdxLista].SlabDimension.XDim 			:= 0;
				ActualPickingListFromHMI[IdxLista].SlabDimension.YDim 			:= 0;
				ActualPickingListFromHMI[IdxLista].SlabDimension.ZDim 			:= 0;
				ActualPickingListFromHMI[IdxLista].SupportPianoLegno 			:= SupportDataEmpty;
				ActualPickingListFromHMI[IdxLista].SupportPianoFerro 			:= SupportDataEmpty;
				ActualPickingListFromHMI[IdxLista].SupportVertBundle 			:= SupportDataEmpty;
				ActualPickingListFromHMI[IdxLista].SupportVertCav 			 	:= SupportDataEmpty;
				
				HMI_ErroreCalcoloLista 		:= 0;
				Cmd_CalcolaLista[IdxLista] 	:= FALSE;
				HMI_Forming_Attivazione[IdxLista] 	:= FALSE;//attivo nuova formatura
				Cmd_AzzeraLista[IdxLista] := FALSE;
				//Ack 
				//IF HMI_ErrAckCalcolaFormatura THEN
					HMI_Forming_ErroreCalcoli := 0;
					HMI_ErrAckCalcolaFormatura := FALSE;
					FOR i:= 1 TO MAXFORMING DO
						HMI_ConfermaAttivazioneFormatura[i] := FALSE;
						HMI_Forming_FormaturaAttivata[i] := FALSE;
					END_FOR
				//END_IF
				CalcolaFormaturaTrig := FALSE;
			END_IF



//--------------------------------------------------------
		// COMANDO ATTIVAZIONE  lista di picking	
//--------------------------------------------------------		 		  
			//Se non ho una Destinazione impostata, Num.pezzi impostato, o Num.pezzi richiesto...
			//	Resetto il comando		
					IF Cmd_AttivaLista[1] = TRUE  THEN
						FOR uu := Iforstart TO Iforend DO
							 	IF	HMI_WorkAreaDataPicking[uu].Typology = CAVALLETTO THEN 
									CASE HMI_WorkAreaDataPicking[uu].TipoTrabajoLado_Cavallete OF 
	 									0:
											HMI_NumeroPezziPresentiPostazione[uu] := HMI_NumeroPezziPresentiCavallete[uu].HMI_NumeroPezziPresentiPostazione_A_Cavaleto +
												 HMI_NumeroPezziPresentiCavallete[uu].HMI_NumeroPezziPresentiPostazione_B_Cavaleto ;
										1:
											HMI_NumeroPezziPresentiPostazione[uu] := HMI_NumeroPezziPresentiCavallete[uu].HMI_NumeroPezziPresentiPostazione_A_Cavaleto ;									 ;
											 
										2:	
		   									HMI_NumeroPezziPresentiPostazione[uu] := HMI_NumeroPezziPresentiCavallete[uu].HMI_NumeroPezziPresentiPostazione_B_Cavaleto ;
												 
									END_CASE
								END_IF 	 
							END_FOR		  
											
													  
																
						IF 	(HMI_WorkAreaDataPicking[1].Destinazione =0 AND 
							HMI_WorkAreaDataPicking[2].Destinazione =0 AND
							HMI_WorkAreaDataPicking[3].Destinazione =0 AND 
							HMI_WorkAreaDataPicking[4].Destinazione =0 AND	 
							HMI_WorkAreaDataPicking[5].Destinazione =0 AND 
							HMI_WorkAreaDataPicking[6].Destinazione =0 AND
							HMI_WorkAreaDataPicking[7].Destinazione =0 AND 
							HMI_WorkAreaDataPicking[8].Destinazione =0)							 
							OR
							(HMI_NumeroPezziPresentiPostazione[1] =0 AND 
							HMI_NumeroPezziPresentiPostazione[2] =0 AND
							HMI_NumeroPezziPresentiPostazione[3] =0 AND 
							HMI_NumeroPezziPresentiPostazione[4] =0 AND
							HMI_NumeroPezziPresentiPostazione[5] =0 AND 
	 						HMI_NumeroPezziPresentiPostazione[6] =0 AND
							HMI_NumeroPezziPresentiPostazione[7] =0 AND 
							HMI_NumeroPezziPresentiPostazione[8] =0)
							OR	 	 
							RequestPickingListFromHMI[1].SlabNumber = 0	 
						THEN
							Cmd_AttivaLista[1] := FALSE;
						 END_IF
					END_IF		  
					IF Cmd_AttivaLista[2] = TRUE  THEN
						FOR uu := Iforstart TO Iforend DO
							 	IF	HMI_WorkAreaDataPicking[uu].Typology = CAVALLETTO THEN 
									CASE HMI_WorkAreaDataPicking[uu].TipoTrabajoLado_Cavallete OF 
	 									0:
											HMI_NumeroPezziPresentiPostazione[uu] := HMI_NumeroPezziPresentiCavallete[uu].HMI_NumeroPezziPresentiPostazione_A_Cavaleto +
												 HMI_NumeroPezziPresentiCavallete[uu].HMI_NumeroPezziPresentiPostazione_B_Cavaleto ;
										1:
											HMI_NumeroPezziPresentiPostazione[uu] := HMI_NumeroPezziPresentiCavallete[uu].HMI_NumeroPezziPresentiPostazione_A_Cavaleto ;									 ;
											 
										2:	
		   									HMI_NumeroPezziPresentiPostazione[uu] := HMI_NumeroPezziPresentiCavallete[uu].HMI_NumeroPezziPresentiPostazione_B_Cavaleto ;
												 
									END_CASE
								END_IF 	 
							END_FOR		  
						IF 	(HMI_WorkAreaDataPicking[1].Destinazione =0 AND 
							HMI_WorkAreaDataPicking[2].Destinazione =0 AND
							HMI_WorkAreaDataPicking[3].Destinazione =0 AND 
							HMI_WorkAreaDataPicking[4].Destinazione =0)
							OR
							(HMI_NumeroPezziPresentiPostazione[1] =0 AND 
							HMI_NumeroPezziPresentiPostazione[2] =0 AND
							HMI_NumeroPezziPresentiPostazione[3] =0 AND 
							HMI_NumeroPezziPresentiPostazione[4] =0)
							OR	 
							RequestPickingListFromHMI[2].SlabNumber = 0	 	 
						THEN
							Cmd_AttivaLista[2] := FALSE;
						 END_IF
					END_IF		
					IF Cmd_AttivaLista[3] = TRUE  THEN
					  FOR uu := Iforstart TO Iforend DO
							 	IF	HMI_WorkAreaDataPicking[uu].Typology = CAVALLETTO THEN 
									CASE HMI_WorkAreaDataPicking[uu].TipoTrabajoLado_Cavallete OF 
	 									0:
											HMI_NumeroPezziPresentiPostazione[uu] := HMI_NumeroPezziPresentiCavallete[uu].HMI_NumeroPezziPresentiPostazione_A_Cavaleto +
												 HMI_NumeroPezziPresentiCavallete[uu].HMI_NumeroPezziPresentiPostazione_B_Cavaleto ;
										1:
											HMI_NumeroPezziPresentiPostazione[uu] := HMI_NumeroPezziPresentiCavallete[uu].HMI_NumeroPezziPresentiPostazione_A_Cavaleto ;									 ;
											 
										2:	
		   									HMI_NumeroPezziPresentiPostazione[uu] := HMI_NumeroPezziPresentiCavallete[uu].HMI_NumeroPezziPresentiPostazione_B_Cavaleto ;
												 
									END_CASE
								END_IF 	 
							END_FOR		  
						IF 	(HMI_WorkAreaDataPicking[5].Destinazione =0 AND 
							HMI_WorkAreaDataPicking[6].Destinazione =0 AND
							HMI_WorkAreaDataPicking[7].Destinazione =0 AND 
							HMI_WorkAreaDataPicking[8].Destinazione =0)
							OR
							(HMI_NumeroPezziPresentiPostazione[5] =0 AND 
							HMI_NumeroPezziPresentiPostazione[6] =0 AND
							HMI_NumeroPezziPresentiPostazione[7] =0 AND 
							HMI_NumeroPezziPresentiPostazione[8] =0)
							OR	 	 
							RequestPickingListFromHMI[3].SlabNumber = 0	 	 
						THEN
							Cmd_AttivaLista[3] := FALSE;
						 END_IF
					END_IF		
{Region "Prmer Bucle cuenta las piezas a coger y rellena el workareastate Con el Tipo Palet"}

			// COMANDO ATTIVAZIONE  lista di picking	
		    IF Cmd_AttivaLista[IdxLista] AND ActualPickingListFromHMI[IdxLista].State <> e_StatoWorkOrder.IN_ESECUZIONE THEN
				ElementiDaDepositare[IdxLista]   :=0;
				HMI_ErroreCalcoloLista := 0;
				HMI_NumeroLastreDepOrdineAttuale[IdxLista] := 0;
				FOR i:= Iforstart TO Iforend DO	
					//HMI_WorkAreaDataPicking[i].Destinazione := FALSE;
					//HMI_WorkAreaDataPicking[i].NumElementiDaLavorare := 0;
					WorkAreaState[i].P := 1;
					WorkAreaProductionList[i] := ListaEmpty;
				END_FOR	 
				
				FOR i:= Iforstart TO Iforend DO	
					IF NOT HMI_WorkAreaDataPicking[i].Destinazione THEN
						ElementiDaDepositare[IdxLista] := ElementiDaDepositare[IdxLista] +HMI_WorkAreaDataPicking[i].NumElementiDaLavorare;
						WorkAreaState[i].P := HMI_WorkAreaDataPicking[i].NumElementiDaLavorare +1;
									   
						CASE HMI_WorkAreaDataPicking[i].Typology OF
							LEGNO_PIANO,TELAIO_PIANO:
								WorkareaState[i].Supporto.Tipologia := e_Tipo_Pallet.CASSA_STANDARD;
							A_FRAME_VERT:	
								WorkareaState[i].Supporto.Tipologia := e_Tipo_Pallet.CAVALLETTO;
								
							IF HMI_WorkAreaDataPicking[i].NumElementiDaLavorare > 0 THEN 
								NuEstacionesPiking := NuEstacionesPiking + 1 ;	
								PosCavalleteOrdenPikin[i]	:=  e_Tipo_Pallet.CAVALLETTO;  
							END_IF
							BUNDLE_VERT:
								WorkareaState[i].Supporto.Tipologia := e_Tipo_Pallet.BUNDLE;	
							
						 ELSE
								WorkareaState[i].Supporto.Tipologia := e_Tipo_Pallet.CASSA_STANDARD;		   
						 END_CASE
					ELSE
						NumPostazioneDeposito := i; NuEstacionPiking := i;
						
						HMI_WorkAreaDataPicking[NumPostazioneDeposito].NumElementiDaLavorare := RequestPickingListFromHMI[IdxLista].SlabNumber;
						CASE HMI_WorkAreaDataPicking[i].Typology OF
							LEGNO_PIANO,TELAIO_PIANO:
								WorkareaState[i].Supporto.Tipologia := e_Tipo_Pallet.CASSA_STANDARD;
							A_FRAME_VERT:	
								WorkareaState[i].Supporto.Tipologia := e_Tipo_Pallet.CAVALLETTO;
								NuEstacionesPiking := NuEstacionesPiking + 1 ;	
								PosCavalleteOrdenPikin[i]	:=  e_Tipo_Pallet.CAVALLETTO;  	 
							BUNDLE_VERT:
								WorkareaState[i].Supporto.Tipologia := e_Tipo_Pallet.BUNDLE;	
								
							
						 ELSE
								WorkareaState[i].Supporto.Tipologia := e_Tipo_Pallet.CASSA_STANDARD;		   
						 END_CASE
					END_IF

		  
//HMI_NumeroPezziPresentiPostazione[i] := WorkAreaState[i].P -1; //NB:cancellato xckè alla attivazione azzerava il num.pezzi presenti sulle postazioni di prelievo
				END_FOR
	
				IF ElementiDaDepositare[IdxLista] <= HMI_WorkAreaDataPicking[NumPostazioneDeposito].NumElementiDaLavorare THEN
					ActualPickingListFromHMI[IdxLista] 				:= RequestPickingListFromHMI[IdxLista];
					ActualPickingListFromHMI[IdxLista].State 		:= e_StatoWorkOrder.DA_ESEGUIRE;

				ELSE
					HMI_ErroreCalcoloLista := 1;
				END_IF
				Cmd_AttivaLista[IdxLista] 				:= FALSE;
				 
			ELSE
				Cmd_AttivaLista[IdxLista] 				:= FALSE;
				 
			END_IF
{endregion}	

{region "Cotas posicione de trabajo"}

//--------------------------------------------------------------------				
//////// attivazione lista di picking : StatoWorkOrder.DA_ESEGUIRE ///
//--------------------------------------------------------------------				
			IF ActualPickingListFromHMI[IdxLista].State = e_StatoWorkOrder.DA_ESEGUIRE  THEN
				ListaInEsecuzione[IdxLista] := FALSE;
				NumeroListaInEsecuzione := 0;
			
				(* Inserimento sequenza di prelievo dalle postazioni in base al quello che l'operatore ha editato da HMI*)
				ElementiDaDepositare[IdxLista] := 0;
				ElementiElaborati[IdxLista]    := 1;
				NumPostazioneDeposito := 0;
				//FOR i:= 1 TO MAXAREAPRESENT DO
				//	WorkAreaState[i].P := 1;
				//END_FOR		
				
				FOR i:= Iforstart TO Iforend DO//---------- For 1 HMI_WorkAreaDataPicking[i].Destinazione 
					IF HMI_WorkAreaDataPicking[i].Destinazione THEN  //-------> Palet destino
						NumPostazioneDeposito := i;
						HMI_WorkAreaDataPicking[NumPostazioneDeposito].NumElementiDaLavorare 	:= RequestPickingListFromHMI[IdxLista].SlabNumber;
						(*CASE HMI_WorkAreaDataPicking[i].Typology OF     // case Pricipal1*)		 
						CASE HMI_WorkAreaDataPicking[NumPostazioneDeposito].Typology OF     // case Pricipal1	
							(* Se ho un legno in piano *)	 
							LEGNO_PIANO:	
								WorkAreaState[NumPostazioneDeposito].Supporto.Code 						:= ActualPickingListFromHMI[IdxLista].SupportPianoLegno.Code;
								WorkAreaState[NumPostazioneDeposito].Supporto.AltezzaDenteRitenuta 		:= ActualPickingListFromHMI[IdxLista].SupportPianoLegno.DimBaseUtile;
								WorkAreaState[NumPostazioneDeposito].Supporto.DimVertice 				:= ActualPickingListFromHMI[IdxLista].SupportPianoLegno.DimVertice;
								WorkAreaState[NumPostazioneDeposito].Supporto.HMAX 						:= ActualPickingListFromHMI[IdxLista].SupportPianoLegno.HMAX;
								WorkAreaState[NumPostazioneDeposito].Supporto.Tipologia 				:= e_Tipo_Pallet.CASSA_STANDARD;//ActualPickingListFromHMI.Support.Tipologia;
								WorkAreaState[NumPostazioneDeposito].Supporto.XDim 						:= ActualPickingListFromHMI[IdxLista].SupportPianoLegno.XDim;
								WorkAreaState[NumPostazioneDeposito].Supporto.YDim 						:= ActualPickingListFromHMI[IdxLista].SupportPianoLegno.YDim;
								WorkAreaState[NumPostazioneDeposito].Supporto.ZDim 						:= ActualPickingListFromHMI[IdxLista].SupportPianoLegno.ZDim;
								WorkAreaOffset[NumPostazioneDeposito].Y 								:= OFFSET_POSTAZIONE_LEGNO + ActualPickingListFromHMI[IdxLista].SupportPianoLegno.YDim/2;//ATTENZIONE!!! per poter lavorare in centro con i supporti pari, questa misura è la distanza tra il riscontro bundle verticale e il centro postazione PARI
								
								CASE HMI_WorkAreaDataPicking[NumPostazioneDeposito].Typology OF
									LEGNO_PIANO:
										 		WorkAreaProductionList[NumPostazioneDeposito].Support := WorkAreaState[NumPostazioneDeposito].Supporto;
												WorkAreaProductionList[NumPostazioneDeposito].Support.Tipologia	:= e_Tipo_Pallet.CASSA_STANDARD; 
									TELAIO_PIANO:
										 		WorkAreaProductionList[NumPostazioneDeposito].Support := WorkAreaState[NumPostazioneDeposito].Supporto;
												WorkAreaProductionList[NumPostazioneDeposito].Support.Tipologia	:= e_Tipo_Pallet.CASSA_STANDARD; 
									BUNDLE_VERT:
										 		WorkAreaProductionList[NumPostazioneDeposito].Support := WorkAreaState[NumPostazioneDeposito].Supporto;
												WorkAreaProductionList[NumPostazioneDeposito].Support.Tipologia	:= e_Tipo_Pallet.BUNDLE; 
												
									A_FRAME_VERT:
										 		WorkAreaProductionList[NumPostazioneDeposito].Support := WorkAreaState[NumPostazioneDeposito].Supporto;
												WorkAreaProductionList[NumPostazioneDeposito].Support.Tipologia	:= e_Tipo_Pallet.CAVALLETTO; 
												
								END_CASE
								FOR j:= Iforstart TO Iforend DO
									IF NOT HMI_WorkAreaDataPicking[j].Destinazione THEN
										IF HMI_WorkAreaDataPicking[j].NumElementiDaLavorare >= 1 THEN
											ElementiDaDepositare[IdxLista] := ElementiElaborati[IdxLista] + HMI_WorkAreaDataPicking[j].NumElementiDaLavorare;
											FOR k := ElementiElaborati[IdxLista] TO ElementiDaDepositare[IdxLista]-1 DO	
												WorkAreaProductionList[NumPostazioneDeposito].PElementList[k].WA_PRELIEVO := j;
												WorkAreaProductionList[NumPostazioneDeposito].PElementList[k].WA_DEPOSITO := i;	
												ElementiElaborati[IdxLista] := ElementiElaborati[IdxLista]+1; 
											END_FOR
											CASE HMI_WorkAreaDataPicking[j].Typology OF 
												(* Se ho una cassa pianale in legno *)
												LEGNO_PIANO:
													WorkAreaState[j].Supporto.Code 					:= ActualPickingListFromHMI[IdxLista].SupportPianoLegno.Code;
													WorkAreaState[j].Supporto.DimBaseUtile		 	:= ActualPickingListFromHMI[IdxLista].SupportPianoLegno.DimBaseUtile;
													WorkAreaState[j].Supporto.AltezzaDenteRitenuta 	:= ActualPickingListFromHMI[IdxLista].SupportPianoLegno.ZDim+20;
													WorkAreaState[j].Supporto.DimVertice 			:= ActualPickingListFromHMI[IdxLista].SupportPianoLegno.DimVertice;
													WorkAreaState[j].Supporto.HMAX 					:= ActualPickingListFromHMI[IdxLista].SupportPianoLegno.HMAX;
													WorkAreaState[j].Supporto.Tipologia 			:= e_Tipo_Pallet.CASSA_STANDARD;//ActualPickingListFromHMI[1].Support.Tipologia;
													WorkAreaState[j].Supporto.XDim 					:= ActualPickingListFromHMI[IdxLista].SupportPianoLegno.XDim;
													WorkAreaState[j].Supporto.YDim 					:= ActualPickingListFromHMI[IdxLista].SupportPianoLegno.YDim;
													WorkAreaState[j].Supporto.ZDim 					:= ActualPickingListFromHMI[IdxLista].SupportPianoLegno.ZDim;
													WorkAreaOffset[j].Y 							:= OFFSET_POSTAZIONE_LEGNO + ActualPickingListFromHMI[IdxLista].SupportPianoLegno.YDim/2;//ATTENZIONE!!! per poter lavorare in centro con i supporti pari, questa misura è la distanza tra il riscontro bundle verticale e il centro postazione PARI
												(* Se ho una cassa pianale in ferro su supporto *)
												TELAIO_PIANO:
													WorkAreaState[j].Supporto.Code 					:= ActualPickingListFromHMI[IdxLista].SupportPianoFerro.Code;
													WorkAreaState[j].Supporto.DimBaseUtile		 	:= ActualPickingListFromHMI[IdxLista].SupportPianoFerro.DimBaseUtile;
													WorkAreaState[j].Supporto.AltezzaDenteRitenuta 	:= ActualPickingListFromHMI[IdxLista].SupportPianoFerro.ZDim+20;
													WorkAreaState[j].Supporto.DimVertice 			:= ActualPickingListFromHMI[IdxLista].SupportPianoFerro.DimVertice;
													WorkAreaState[j].Supporto.HMAX 					:= ActualPickingListFromHMI[IdxLista].SupportPianoFerro.HMAX;
													WorkAreaState[j].Supporto.Tipologia 			:=  e_Tipo_Pallet.CASSA_STANDARD;//ActualPickingListFromHMI[1].Support.Tipologia;
													WorkAreaState[j].Supporto.XDim 					:= ActualPickingListFromHMI[IdxLista].SupportPianoFerro.XDim;
													WorkAreaState[j].Supporto.YDim 					:= ActualPickingListFromHMI[IdxLista].SupportPianoFerro.YDim;
													WorkAreaState[j].Supporto.ZDim 					:= ActualPickingListFromHMI[IdxLista].SupportPianoFerro.ZDim;
													WorkAreaOffset[j].Y 							:= OFFSET_POSTAZIONE_TELAIO - ActualPickingListFromHMI[IdxLista].SupportPianoFerro.YDim/2;//ATTENZIONE!!! per poter lavorare in centro con i supporti pari, questa misura è la distanza tra il riscontro bundle verticale e il centro postazione PARI
												(* Se ho un bundle *)
												BUNDLE_VERT:
													//WorkAreaState[j].P := ElementiDaDepositare;
													WorkAreaState[j].Supporto.Code 					:= ActualPickingListFromHMI[IdxLista].SupportVertBundle.Code;
													WorkAreaState[j].Supporto.DimBaseUtile		 	:= ActualPickingListFromHMI[IdxLista].SupportVertBundle.DimBaseUtile;
													WorkAreaState[j].Supporto.AltezzaDenteRitenuta 	:= ActualPickingListFromHMI[IdxLista].SupportVertBundle.ZDim+20;
													WorkAreaState[j].Supporto.DimVertice 			:= ActualPickingListFromHMI[IdxLista].SupportVertBundle.DimVertice;
													WorkAreaState[j].Supporto.HMAX 					:= ActualPickingListFromHMI[IdxLista].SupportVertBundle.HMAX;
													WorkAreaState[j].Supporto.Tipologia 			:= e_Tipo_Pallet.BUNDLE;//ActualPickingListFromHMI.SupportVert.Tipologia;
													WorkAreaState[j].Supporto.XDim 					:= ActualPickingListFromHMI[IdxLista].SupportVertBundle.XDim;
													WorkAreaState[j].Supporto.YDim 					:= ActualPickingListFromHMI[IdxLista].SupportVertBundle.YDim;
													WorkAreaState[j].Supporto.ZDim 					:= ActualPickingListFromHMI[IdxLista].SupportVertBundle.ZDim;
													WorkAreaState[j].Supporto.ZDim_Ext1        		:= WorkAreaState[j].Supporto.ZDim + 20;
													//Lo que HABIA	
													//WorkAreaOffset[j].Y 							:= HMI_OffsetDepositoLastra.Y180 ;
													//Mod 25/&/2025	  
													WorkAreaOffset[NumPostazioneDeposito].Y 		:= ActualPickingListFromHMI[IdxLista].SupportVertBundle.YDim-ActualPickingListFromHMI[IdxLista].SupportVertBundle.DimBaseUtile -40 ;			
												(* Se ho un A_Frame *)	  
												A_FRAME_VERT:  						
													//WorkAreaState[j].P := ElementiDaDepositare;
													WorkAreaState[j].Supporto.Code 					:= ActualPickingListFromHMI[IdxLista].SupportVertCav.Code;
													WorkAreaState[j].Supporto.DimBaseUtile		 	:= ActualPickingListFromHMI[IdxLista].SupportVertCav.DimBaseUtile;
													WorkAreaState[j].Supporto.AltezzaDenteRitenuta 	:= ActualPickingListFromHMI[IdxLista].SupportVertCav.ZDim+20;
													WorkAreaState[j].Supporto.DimVertice 			:= ActualPickingListFromHMI[IdxLista].SupportVertCav.DimVertice;
													WorkAreaState[j].Supporto.HMAX 					:= ActualPickingListFromHMI[IdxLista].SupportVertCav.HMAX;
													WorkAreaState[j].Supporto.Tipologia 			:= CAVALLETTO;//ActualPickingListFromHMI.SupportVertCav.Tipologia;
													WorkAreaState[j].Supporto.XDim 					:= ActualPickingListFromHMI[IdxLista].SupportVertCav.XDim;
													WorkAreaState[j].Supporto.YDim 					:= ActualPickingListFromHMI[IdxLista].SupportVertCav.YDim;
													WorkAreaState[j].Supporto.ZDim 					:= ActualPickingListFromHMI[IdxLista].SupportVertCav.ZDim;
													WorkAreaState[j].Supporto.ZDim_Ext1        		:= WorkAreaState[j].Supporto.ZDim + 20;	
													WorkAreaState[j].Supporto.TipoTrabajoLado_Cavallete := HMI_WorkAreaDataPicking[j].TipoTrabajoLado_Cavallete ;	
													WorkAreaOffset[j].Y 							:= OFFSET_POSTAZIONE_LEGNO + ActualPickingListFromHMI[IdxLista].SupportVertCav.YDim/2;//ATTENZIONE!!! per poter lavorare in centro con i supporti pari, questa misura è la distanza tra il riscontro bundle verticale e il centro postazione PARI
											   		CoordenadaPasillo0_Y := WorkArea[j].Y +  WorkAreaOffset[j].Y  - Dimensioni_Pinza.Spessore - INGOMBRO_RISCONTRO_BUNDLE - WorkAreaState[j].Supporto.YDim /2 ;
													CoordenadaPasillo180_Y := WorkArea[j].Y + WorkAreaState[j].Supporto.YDim /2 + WorkAreaOffset[j].Y  + Dimensioni_Pinza.Spessore + INGOMBRO_RISCONTRO_FRAME  ;	
											END_CASE	
											WorkAreaProductionList[j].Support := HMI_Formatura.HMI_Forming_Supporto; 
										END_IF
									END_IF     
									TFClearApprendimento(ADR(WorkAreaState[j].Apprendimento));//Azzeramento apprendimento 
								END_FOR
								EXIT; 
							(* Se ho un telaio in piano *)	 
							TELAIO_PIANO:	
								WorkAreaState[NumPostazioneDeposito].Supporto.Code 						:= ActualPickingListFromHMI[IdxLista].SupportPianoFerro.Code;
								WorkAreaState[NumPostazioneDeposito].Supporto.AltezzaDenteRitenuta 		:= ActualPickingListFromHMI[IdxLista].SupportPianoFerro.DimBaseUtile;
								WorkAreaState[NumPostazioneDeposito].Supporto.DimVertice 				:= ActualPickingListFromHMI[IdxLista].SupportPianoFerro.DimVertice;
								WorkAreaState[NumPostazioneDeposito].Supporto.HMAX 						:= ActualPickingListFromHMI[IdxLista].SupportPianoFerro.HMAX;
								WorkAreaState[NumPostazioneDeposito].Supporto.Tipologia 				:= CASSA_STANDARD;//ActualPickingListFromHMI.Support.Tipologia;
								WorkAreaState[NumPostazioneDeposito].Supporto.XDim 						:= ActualPickingListFromHMI[IdxLista].SupportPianoFerro.XDim;
								WorkAreaState[NumPostazioneDeposito].Supporto.YDim 						:= ActualPickingListFromHMI[IdxLista].SupportPianoFerro.YDim;
								WorkAreaState[NumPostazioneDeposito].Supporto.ZDim 						:= ActualPickingListFromHMI[IdxLista].SupportPianoFerro.ZDim;
								WorkAreaOffset[NumPostazioneDeposito].Y 								:= OFFSET_POSTAZIONE_TELAIO - ActualPickingListFromHMI[IdxLista].SupportPianoFerro.YDim/2;//ATTENZIONE!!! per poter lavorare in centro con i supporti pari, questa misura è la distanza tra il riscontro bundle verticale e il centro postazione PARI
								CASE HMI_WorkAreaDataPicking[NumPostazioneDeposito].Typology OF
									LEGNO_PIANO:
										 		WorkAreaProductionList[NumPostazioneDeposito].Support := WorkAreaState[NumPostazioneDeposito].Supporto;
												WorkAreaProductionList[NumPostazioneDeposito].Support.Tipologia	:= e_Tipo_Pallet.CASSA_STANDARD; 
									TELAIO_PIANO:
										 		WorkAreaProductionList[NumPostazioneDeposito].Support := WorkAreaState[NumPostazioneDeposito].Supporto;
												WorkAreaProductionList[NumPostazioneDeposito].Support.Tipologia	:= e_Tipo_Pallet.CASSA_STANDARD; 
									BUNDLE_VERT:
										 		WorkAreaProductionList[NumPostazioneDeposito].Support := WorkAreaState[NumPostazioneDeposito].Supporto;
												WorkAreaProductionList[NumPostazioneDeposito].Support.Tipologia	:= e_Tipo_Pallet.BUNDLE; 
									A_FRAME_VERT:
										 		WorkAreaProductionList[NumPostazioneDeposito].Support := WorkAreaState[NumPostazioneDeposito].Supporto;
												WorkAreaProductionList[NumPostazioneDeposito].Support.Tipologia	:= e_Tipo_Pallet.CAVALLETTO; 
								END_CASE
								
								FOR j:= Iforstart TO Iforend DO
									IF NOT HMI_WorkAreaDataPicking[j].Destinazione THEN
										IF HMI_WorkAreaDataPicking[j].NumElementiDaLavorare >= 1 THEN
											ElementiDaDepositare[IdxLista] := ElementiElaborati[IdxLista] + HMI_WorkAreaDataPicking[j].NumElementiDaLavorare;
											FOR k := ElementiElaborati[IdxLista] TO ElementiDaDepositare[IdxLista]-1 DO	
												WorkAreaProductionList[NumPostazioneDeposito].PElementList[k].WA_PRELIEVO := j;
												WorkAreaProductionList[NumPostazioneDeposito].PElementList[k].WA_DEPOSITO := i;	
												ElementiElaborati[IdxLista] := ElementiElaborati[IdxLista]+1; 
											END_FOR
											CASE HMI_WorkAreaDataPicking[j].Typology OF 
												(* Se ho una cassa pianale in legno *)
												LEGNO_PIANO:
													WorkAreaState[j].Supporto.Code 					:= ActualPickingListFromHMI[IdxLista].SupportPianoLegno.Code;
													WorkAreaState[j].Supporto.DimBaseUtile		 	:= ActualPickingListFromHMI[IdxLista].SupportPianoLegno.DimBaseUtile;
													WorkAreaState[j].Supporto.AltezzaDenteRitenuta 	:= ActualPickingListFromHMI[IdxLista].SupportPianoLegno.ZDim+20;
													WorkAreaState[j].Supporto.DimVertice 			:= ActualPickingListFromHMI[IdxLista].SupportPianoLegno.DimVertice;
													WorkAreaState[j].Supporto.HMAX 					:= ActualPickingListFromHMI[IdxLista].SupportPianoLegno.HMAX;
													WorkAreaState[j].Supporto.Tipologia 			:=  e_Tipo_Pallet.CASSA_STANDARD;//ActualPickingListFromHMI[1].Support.Tipologia;
													WorkAreaState[j].Supporto.XDim 					:= ActualPickingListFromHMI[IdxLista].SupportPianoLegno.XDim;
													WorkAreaState[j].Supporto.YDim 					:= ActualPickingListFromHMI[IdxLista].SupportPianoLegno.YDim;
													WorkAreaState[j].Supporto.ZDim 					:= ActualPickingListFromHMI[IdxLista].SupportPianoLegno.ZDim;
													WorkAreaOffset[j].Y 							:= OFFSET_POSTAZIONE_LEGNO + ActualPickingListFromHMI[IdxLista].SupportPianoLegno.YDim/2;//ATTENZIONE!!! per poter lavorare in centro con i supporti pari, questa misura è la distanza tra il riscontro bundle verticale e il centro postazione PARI
												(* Se ho una cassa pianale in ferro su supporto *)
												TELAIO_PIANO:
													WorkAreaState[j].Supporto.Code 					:= ActualPickingListFromHMI[IdxLista].SupportPianoFerro.Code;
													WorkAreaState[j].Supporto.DimBaseUtile		 	:= ActualPickingListFromHMI[IdxLista].SupportPianoFerro.DimBaseUtile;
													WorkAreaState[j].Supporto.AltezzaDenteRitenuta 	:= ActualPickingListFromHMI[IdxLista].SupportPianoFerro.ZDim+20;
													WorkAreaState[j].Supporto.DimVertice 			:= ActualPickingListFromHMI[IdxLista].SupportPianoFerro.DimVertice;
													WorkAreaState[j].Supporto.HMAX 					:= ActualPickingListFromHMI[IdxLista].SupportPianoFerro.HMAX;
													WorkAreaState[j].Supporto.Tipologia 			:=  e_Tipo_Pallet.CASSA_STANDARD;//ActualPickingListFromHMI[1].Support.Tipologia;
													WorkAreaState[j].Supporto.XDim 					:= ActualPickingListFromHMI[IdxLista].SupportPianoFerro.XDim;
													WorkAreaState[j].Supporto.YDim 					:= ActualPickingListFromHMI[IdxLista].SupportPianoFerro.YDim;
													WorkAreaState[j].Supporto.ZDim 					:= ActualPickingListFromHMI[IdxLista].SupportPianoFerro.ZDim;
													WorkAreaOffset[j].Y 							:= OFFSET_POSTAZIONE_TELAIO - ActualPickingListFromHMI[IdxLista].SupportPianoFerro.YDim/2;//ATTENZIONE!!! per poter lavorare in centro con i supporti pari, questa misura è la distanza tra il riscontro bundle verticale e il centro postazione PARI
												(* Se ho un bundle *)
												BUNDLE_VERT:
													//WorkAreaState[j].P := ElementiDaDepositare;
													WorkAreaState[j].Supporto.Code 					:= ActualPickingListFromHMI[IdxLista].SupportVertBundle.Code;
													WorkAreaState[j].Supporto.DimBaseUtile		 	:= ActualPickingListFromHMI[IdxLista].SupportVertBundle.DimBaseUtile;
													WorkAreaState[j].Supporto.AltezzaDenteRitenuta 	:= ActualPickingListFromHMI[IdxLista].SupportVertBundle.ZDim+20;
													WorkAreaState[j].Supporto.DimVertice 			:= ActualPickingListFromHMI[IdxLista].SupportVertBundle.DimVertice;
													WorkAreaState[j].Supporto.HMAX 					:= ActualPickingListFromHMI[IdxLista].SupportVertBundle.HMAX;
													WorkAreaState[j].Supporto.Tipologia 			:= e_Tipo_Pallet.BUNDLE;//ActualPickingListFromHMI.SupportVertBundle.Tipologia;
													WorkAreaState[j].Supporto.XDim 					:= ActualPickingListFromHMI[IdxLista].SupportVertBundle.XDim;
													WorkAreaState[j].Supporto.YDim 					:= ActualPickingListFromHMI[IdxLista].SupportVertBundle.YDim;
													WorkAreaState[j].Supporto.ZDim 					:= ActualPickingListFromHMI[IdxLista].SupportVertBundle.ZDim;
													WorkAreaState[j].Supporto.ZDim_Ext1        		:= WorkAreaState[j].Supporto.ZDim + 20;	
													 WorkAreaOffset[j].Y 		:= 0 ;	
													//Mod 25/&/2025	  
													//WorkAreaOffset[j].Y 		:= ActualPickingListFromHMI[IdxLista].SupportVertBundle.YDim-ActualPickingListFromHMI[IdxLista].SupportVertBundle.DimBaseUtile -40;				
												(* Se ho un A_Frame *)	  
												A_FRAME_VERT:  						
													//WorkAreaState[j].P := ElementiDaDepositare;
													WorkAreaState[j].Supporto.Code 					:= ActualPickingListFromHMI[IdxLista].SupportVertCav.Code;
													WorkAreaState[j].Supporto.DimBaseUtile		 	:= ActualPickingListFromHMI[IdxLista].SupportVertCav.DimBaseUtile;
													WorkAreaState[j].Supporto.AltezzaDenteRitenuta 	:= ActualPickingListFromHMI[IdxLista].SupportVertCav.ZDim+20;
													WorkAreaState[j].Supporto.DimVertice 			:= ActualPickingListFromHMI[IdxLista].SupportVertCav.DimVertice;
													WorkAreaState[j].Supporto.HMAX 					:= ActualPickingListFromHMI[IdxLista].SupportVertcav.HMAX;
													WorkAreaState[j].Supporto.Tipologia 			:= CAVALLETTO;//ActualPickingListFromHMI.SupportVert.Tipologia;
													WorkAreaState[j].Supporto.XDim 					:= ActualPickingListFromHMI[IdxLista].SupportVertCav.XDim;
													WorkAreaState[j].Supporto.YDim 					:= ActualPickingListFromHMI[IdxLista].SupportVertCav.YDim;
													WorkAreaState[j].Supporto.ZDim 					:= ActualPickingListFromHMI[IdxLista].SupportVertCav.ZDim;
													WorkAreaState[j].Supporto.ZDim_Ext1        		:= WorkAreaState[j].Supporto.ZDim + 20;	
													WorkAreaState[j].Supporto.TipoTrabajoLado_Cavallete := HMI_WorkAreaDataPicking[j].TipoTrabajoLado_Cavallete ;	
													WorkAreaOffset[j].Y 							:= OFFSET_POSTAZIONE_LEGNO + ActualPickingListFromHMI[IdxLista].SupportVertCav.YDim/2;//ATTENZIONE!!! per poter lavorare in centro con i supporti pari, questa misura è la distanza tra il riscontro bundle verticale e il centro postazione PARI
											   		CoordenadaPasillo0_Y := WorkArea[j].Y +  WorkAreaOffset[j].Y  - Dimensioni_Pinza.Spessore - INGOMBRO_RISCONTRO_BUNDLE - WorkAreaState[j].Supporto.YDim /2 ;
													CoordenadaPasillo180_Y := WorkArea[j].Y + WorkAreaState[j].Supporto.YDim /2 + WorkAreaOffset[j].Y  + Dimensioni_Pinza.Spessore + INGOMBRO_RISCONTRO_FRAME  ;	
											END_CASE	
											WorkAreaProductionList[j].Support := HMI_Formatura.HMI_Forming_Supporto; 
										END_IF
									END_IF     
									TFClearApprendimento(ADR(WorkAreaState[j].Apprendimento));//Azzeramento apprendimento 
								END_FOR
								EXIT; 
							(* Se ho un bundle *)
							BUNDLE_VERT:
								CASE HMI_WorkAreaDataPicking[NumPostazioneDeposito].Typology OF
									LEGNO_PIANO:
										 		WorkAreaProductionList[NumPostazioneDeposito].Support := WorkAreaState[NumPostazioneDeposito].Supporto;
												WorkAreaProductionList[NumPostazioneDeposito].Support.Tipologia	:= e_Tipo_Pallet.CASSA_STANDARD; 
									TELAIO_PIANO:
										 		WorkAreaProductionList[NumPostazioneDeposito].Support := WorkAreaState[NumPostazioneDeposito].Supporto;
												WorkAreaProductionList[NumPostazioneDeposito].Support.Tipologia	:= e_Tipo_Pallet.CASSA_STANDARD; 
									BUNDLE_VERT:
										 		WorkAreaProductionList[NumPostazioneDeposito].Support := WorkAreaState[NumPostazioneDeposito].Supporto;
												WorkAreaProductionList[NumPostazioneDeposito].Support.Tipologia	:= e_Tipo_Pallet.BUNDLE; 
									A_FRAME_VERT:
										 		WorkAreaProductionList[NumPostazioneDeposito].Support := WorkAreaState[NumPostazioneDeposito].Supporto;
												WorkAreaProductionList[NumPostazioneDeposito].Support.Tipologia	:= e_Tipo_Pallet.CAVALLETTO; 
								END_CASE
								//Se ho deposito verticale su bundle
								WorkAreaState[NumPostazioneDeposito].Supporto.Code 						:= ActualPickingListFromHMI[IdxLista].SupportVertBundle.Code;
								WorkAreaState[NumPostazioneDeposito].Supporto.DimBaseUtile		 		:= ActualPickingListFromHMI[IdxLista].SupportVertBundle.DimBaseUtile;
								WorkAreaState[NumPostazioneDeposito].Supporto.DimVertice 				:= ActualPickingListFromHMI[IdxLista].SupportVertBundle.DimVertice;
								WorkAreaState[NumPostazioneDeposito].Supporto.HMAX 						:= ActualPickingListFromHMI[IdxLista].SupportVertBundle.HMAX;
								WorkAreaState[NumPostazioneDeposito].Supporto.Tipologia 				:= e_Tipo_Pallet.BUNDLE;
								WorkAreaState[NumPostazioneDeposito].Supporto.XDim 						:= ActualPickingListFromHMI[IdxLista].SupportVertBundle.XDim;
								WorkAreaState[NumPostazioneDeposito].Supporto.YDim 						:= ActualPickingListFromHMI[IdxLista].SupportVertBundle.YDim;
								WorkAreaState[NumPostazioneDeposito].Supporto.ZDim 						:= ActualPickingListFromHMI[IdxLista].SupportVertBundle.ZDim;
								//Lo que HABIA
								//PruevaWorkAreaOffset[NumPostazioneDeposito].Y 								:= -40;	
								//Mod 25/&/2025	  
								//WorkAreaOffset[NumPostazioneDeposito].Y 								:= ActualPickingListFromHMI[IdxLista].SupportVertBundle.YDim-ActualPickingListFromHMI[IdxLista].SupportVertBundle.DimBaseUtile -20;
								FOR j:= Iforstart TO Iforend DO
									IF NOT HMI_WorkAreaDataPicking[j].Destinazione THEN
										IF HMI_WorkAreaDataPicking[j].NumElementiDaLavorare >= 1 THEN
											ElementiDaDepositare[IdxLista] := ElementiElaborati[IdxLista] + HMI_WorkAreaDataPicking[j].NumElementiDaLavorare;
											FOR k := ElementiElaborati[IdxLista] TO ElementiDaDepositare[IdxLista]-1 DO	
												WorkAreaProductionList[NumPostazioneDeposito].PElementList[k].WA_PRELIEVO := j;
												WorkAreaProductionList[NumPostazioneDeposito].PElementList[k].WA_DEPOSITO := i;	
												ElementiElaborati[IdxLista] := ElementiElaborati[IdxLista]+1; 
											END_FOR
											CASE HMI_WorkAreaDataPicking[j].Typology OF 
												(* Se ho una cassa pianale in legno *)
												LEGNO_PIANO:
													WorkAreaState[j].Supporto.Code 					:= ActualPickingListFromHMI[IdxLista].SupportPianoLegno.Code;
													WorkAreaState[j].Supporto.DimBaseUtile		 	:= ActualPickingListFromHMI[IdxLista].SupportPianoLegno.DimBaseUtile;
													WorkAreaState[j].Supporto.AltezzaDenteRitenuta 	:= ActualPickingListFromHMI[IdxLista].SupportPianoLegno.ZDim+20;
													WorkAreaState[j].Supporto.DimVertice 			:= ActualPickingListFromHMI[IdxLista].SupportPianoLegno.DimVertice;
													WorkAreaState[j].Supporto.HMAX 					:= ActualPickingListFromHMI[IdxLista].SupportPianoLegno.HMAX;
													WorkAreaState[j].Supporto.Tipologia 			:=  e_Tipo_Pallet.CASSA_STANDARD;//ActualPickingListFromHMI[1].Support.Tipologia;
													WorkAreaState[j].Supporto.XDim 					:= ActualPickingListFromHMI[IdxLista].SupportPianoLegno.XDim;
													WorkAreaState[j].Supporto.YDim 					:= ActualPickingListFromHMI[IdxLista].SupportPianoLegno.YDim;
													WorkAreaState[j].Supporto.ZDim 					:= ActualPickingListFromHMI[IdxLista].SupportPianoLegno.ZDim;
													WorkAreaOffset[j].Y 							:= OFFSET_POSTAZIONE_LEGNO + ActualPickingListFromHMI[IdxLista].SupportPianoLegno.YDim/2;//ATTENZIONE!!! per poter lavorare in centro con i supporti pari, questa misura è la distanza tra il riscontro bundle verticale e il centro postazione PARI
												(* Se ho una cassa pianale in ferro su supporto *)
												TELAIO_PIANO:
													WorkAreaState[j].Supporto.Code 					:= ActualPickingListFromHMI[IdxLista].SupportPianoFerro.Code;
													WorkAreaState[j].Supporto.DimBaseUtile		 	:= ActualPickingListFromHMI[IdxLista].SupportPianoFerro.DimBaseUtile;
													WorkAreaState[j].Supporto.AltezzaDenteRitenuta 	:= ActualPickingListFromHMI[IdxLista].SupportPianoFerro.ZDim+20;
													WorkAreaState[j].Supporto.DimVertice 			:= ActualPickingListFromHMI[IdxLista].SupportPianoFerro.DimVertice;
													WorkAreaState[j].Supporto.HMAX 					:= ActualPickingListFromHMI[IdxLista].SupportPianoFerro.HMAX;
													WorkAreaState[j].Supporto.Tipologia 			:=  e_Tipo_Pallet.CASSA_STANDARD;//ActualPickingListFromHMI[1].Support.Tipologia;
													WorkAreaState[j].Supporto.XDim 					:= ActualPickingListFromHMI[IdxLista].SupportPianoFerro.XDim;
													WorkAreaState[j].Supporto.YDim 					:= ActualPickingListFromHMI[IdxLista].SupportPianoFerro.YDim;
													WorkAreaState[j].Supporto.ZDim 					:= ActualPickingListFromHMI[IdxLista].SupportPianoFerro.ZDim;
													WorkAreaOffset[j].Y 							:= OFFSET_POSTAZIONE_TELAIO - ActualPickingListFromHMI[IdxLista].SupportPianoFerro.YDim/2;//ATTENZIONE!!! per poter lavorare in centro con i supporti pari, questa misura è la distanza tra il riscontro bundle verticale e il centro postazione PARI
												(* Se ho un bundle *)
												BUNDLE_VERT:
													//WorkAreaState[j].P := ElementiDaDepositare;
													WorkAreaState[j].Supporto.Code 					:= ActualPickingListFromHMI[IdxLista].SupportVertBundle.Code;
													WorkAreaState[j].Supporto.DimBaseUtile		 	:= ActualPickingListFromHMI[IdxLista].SupportVertBundle.DimBaseUtile;
													WorkAreaState[j].Supporto.AltezzaDenteRitenuta 	:= ActualPickingListFromHMI[IdxLista].SupportVertBundle.ZDim+20;
													WorkAreaState[j].Supporto.DimVertice 			:= ActualPickingListFromHMI[IdxLista].SupportVertBundle.DimVertice;
													WorkAreaState[j].Supporto.HMAX 					:= ActualPickingListFromHMI[IdxLista].SupportVertBundle.HMAX;
													WorkAreaState[j].Supporto.Tipologia 			:= e_Tipo_Pallet.BUNDLE;//ActualPickingListFromHMI.SupportVert.Tipologia;
													WorkAreaState[j].Supporto.XDim 					:= ActualPickingListFromHMI[IdxLista].SupportVertBundle.XDim;
													WorkAreaState[j].Supporto.YDim 					:= ActualPickingListFromHMI[IdxLista].SupportVertBundle.YDim;
													WorkAreaState[j].Supporto.ZDim 					:= ActualPickingListFromHMI[IdxLista].SupportVertBundle.ZDim;
													WorkAreaState[j].Supporto.ZDim_Ext1        		:= WorkAreaState[j].Supporto.ZDim + 20;	
													// **Lo Que Habia	
													WorkAreaOffset[j].Y 							:= 0;
													//Mod 25/&/2025	  
													//WorkAreaOffset[j].Y 		:= ActualPickingListFromHMI[IdxLista].SupportVertBundle.YDim-ActualPickingListFromHMI[IdxLista].SupportVertBundle.DimBaseUtile -40;	
			
												(* Se ho un A_Frame *)	  
												A_FRAME_VERT:  						
													//WorkAreaState[j].P := ElementiDaDepositare;
													WorkAreaState[j].Supporto.Code 					:= ActualPickingListFromHMI[IdxLista].SupportVertCav.Code;
													WorkAreaState[j].Supporto.DimBaseUtile		 	:= ActualPickingListFromHMI[IdxLista].SupportVertCav.DimBaseUtile;
													WorkAreaState[j].Supporto.AltezzaDenteRitenuta 	:= ActualPickingListFromHMI[IdxLista].SupportVertCav.ZDim+20;
													WorkAreaState[j].Supporto.DimVertice 			:= ActualPickingListFromHMI[IdxLista].SupportVertCav.DimVertice;
													WorkAreaState[j].Supporto.HMAX 					:= ActualPickingListFromHMI[IdxLista].SupportVertCav.HMAX;
													WorkAreaState[j].Supporto.Tipologia 			:= CAVALLETTO;//ActualPickingListFromHMI.SupportVert.Tipologia;
													WorkAreaState[j].Supporto.XDim 					:= ActualPickingListFromHMI[IdxLista].SupportVertCav.XDim;
													WorkAreaState[j].Supporto.YDim 					:= ActualPickingListFromHMI[IdxLista].SupportVertCav.YDim;
													WorkAreaState[j].Supporto.ZDim 					:= ActualPickingListFromHMI[IdxLista].SupportVertCav.ZDim;
													WorkAreaState[j].Supporto.ZDim_Ext1        		:= WorkAreaState[j].Supporto.ZDim + 20;	
													WorkAreaState[j].Supporto.TipoTrabajoLado_Cavallete := HMI_WorkAreaDataPicking[j].TipoTrabajoLado_Cavallete ;	
													WorkAreaOffset[j].Y 							:= OFFSET_POSTAZIONE_LEGNO + ActualPickingListFromHMI[IdxLista].SupportVertCav.YDim/2;//ATTENZIONE!!! per poter lavorare in centro con i supporti pari, questa misura è la distanza tra il riscontro bundle verticale e il centro postazione PARI
													CoordenadaPasillo0_Y := WorkArea[j].Y +  WorkAreaOffset[j].Y  - Dimensioni_Pinza.Spessore - INGOMBRO_RISCONTRO_BUNDLE - WorkAreaState[j].Supporto.YDim /2 ;
													CoordenadaPasillo180_Y := WorkArea[j].Y + WorkAreaState[j].Supporto.YDim /2 + WorkAreaOffset[j].Y  + Dimensioni_Pinza.Spessore + INGOMBRO_RISCONTRO_FRAME  ;		  
											END_CASE
											//WorkAreaProductionList[j].Support := HMI_Formatura.HMI_Forming_Supporto;		  
											WorkAreaProductionList[j].Support := WorkAreaState[j].Supporto;
										END_IF
									END_IF
									TFClearApprendimento(ADR(WorkAreaState[j].Apprendimento));//Azzeramento apprendimento
								END_FOR
								EXIT; 
							(* Se ho un A_Frame *)	
							A_FRAME_VERT:
								WorkAreaState[NumPostazioneDeposito].Supporto.Code 						:= ActualPickingListFromHMI[IdxLista].SupportVertCav.Code;
								WorkAreaState[NumPostazioneDeposito].Supporto.DimBaseUtile		 		:= ActualPickingListFromHMI[IdxLista].SupportVertCav.DimBaseUtile;
								WorkAreaState[NumPostazioneDeposito].Supporto.DimVertice 				:= ActualPickingListFromHMI[IdxLista].SupportVertCav.DimVertice;
								WorkAreaState[NumPostazioneDeposito].Supporto.HMAX 						:= ActualPickingListFromHMI[IdxLista].SupportVertCav.HMAX;
								WorkAreaState[NumPostazioneDeposito].Supporto.Tipologia 				:= e_Tipo_Pallet.CAVALLETTO;//ActualPickingListFromHMI.SupportVertBundle.Tipologia;
								WorkAreaState[NumPostazioneDeposito].Supporto.XDim 						:= ActualPickingListFromHMI[IdxLista].SupportVertCav.XDim;
								WorkAreaState[NumPostazioneDeposito].Supporto.YDim 						:= ActualPickingListFromHMI[IdxLista].SupportVertCav.YDim;
								WorkAreaState[NumPostazioneDeposito].Supporto.ZDim 						:= ActualPickingListFromHMI[IdxLista].SupportVertCav.ZDim;
								//WorkAreaOffset[NumPostazioneDeposito].Y 								:= OFFSET_POSTAZIONE_LEGNO (*- ActualPickingListFromHMI[IdxLista].SupportPianoFerro.YDim/2*);
								WorkAreaOffset[NumPostazioneDeposito].Y 								:= OFFSET_POSTAZIONE_LEGNO + ActualPickingListFromHMI[IdxLista].SupportVertCav.YDim/2;	
								WorkAreaState[NumPostazioneDeposito].Supporto.TipoTrabajoLado_Cavallete := HMI_WorkAreaDataPicking[NumPostazioneDeposito].TipoTrabajoLado_Cavallete ;
								CASE HMI_WorkAreaDataPicking[NumPostazioneDeposito].Typology OF
									LEGNO_PIANO:
										 		WorkAreaProductionList[NumPostazioneDeposito].Support := WorkAreaState[NumPostazioneDeposito].Supporto;
												WorkAreaProductionList[NumPostazioneDeposito].Support.Tipologia	:= e_Tipo_Pallet.CASSA_STANDARD; 
									TELAIO_PIANO:
										 		WorkAreaProductionList[NumPostazioneDeposito].Support := WorkAreaState[NumPostazioneDeposito].Supporto;
												WorkAreaProductionList[NumPostazioneDeposito].Support.Tipologia	:= e_Tipo_Pallet.CASSA_STANDARD; 
									BUNDLE_VERT:
										 		WorkAreaProductionList[NumPostazioneDeposito].Support := WorkAreaState[NumPostazioneDeposito].Supporto;
												WorkAreaProductionList[NumPostazioneDeposito].Support.Tipologia	:= e_Tipo_Pallet.BUNDLE; 
									A_FRAME_VERT:
										 		WorkAreaProductionList[NumPostazioneDeposito].Support := WorkAreaState[NumPostazioneDeposito].Supporto;
												WorkAreaProductionList[NumPostazioneDeposito].Support.Tipologia	:= e_Tipo_Pallet.CAVALLETTO; 
												CoordenadaPasillo0_Y := WorkArea[NumPostazioneDeposito].Y +  WorkAreaOffset[NumPostazioneDeposito].Y  - Dimensioni_Pinza.Spessore - INGOMBRO_RISCONTRO_BUNDLE - WorkAreaState[NumPostazioneDeposito].Supporto.YDim /2;
												CoordenadaPasillo180_Y := WorkArea[NumPostazioneDeposito].Y + WorkAreaState[NumPostazioneDeposito].Supporto.YDim /2 + WorkAreaOffset[NumPostazioneDeposito].Y  + Dimensioni_Pinza.Spessore + INGOMBRO_RISCONTRO_FRAME  ;		
					  
								END_CASE
								FOR j:= Iforstart TO Iforend DO
									IF NOT HMI_WorkAreaDataPicking[j].Destinazione THEN
										IF HMI_WorkAreaDataPicking[j].NumElementiDaLavorare >= 1 THEN
											ElementiDaDepositare[IdxLista] := ElementiElaborati[IdxLista] + HMI_WorkAreaDataPicking[j].NumElementiDaLavorare;
											FOR k := ElementiElaborati[IdxLista] TO ElementiDaDepositare[IdxLista]-1 DO	
												WorkAreaProductionList[NumPostazioneDeposito].PElementList[k].WA_PRELIEVO := j;
												WorkAreaProductionList[NumPostazioneDeposito].PElementList[k].WA_DEPOSITO := i;	
												ElementiElaborati[IdxLista] := ElementiElaborati[IdxLista]+1; 
											END_FOR
											CASE HMI_WorkAreaDataPicking[j].Typology OF 
												(* Se ho una cassa pianale in legno *)
												LEGNO_PIANO:
													WorkAreaState[j].Supporto.Code 					:= ActualPickingListFromHMI[IdxLista].SupportPianoLegno.Code;
													WorkAreaState[j].Supporto.DimBaseUtile		 	:= ActualPickingListFromHMI[IdxLista].SupportPianoLegno.DimBaseUtile;
													WorkAreaState[j].Supporto.AltezzaDenteRitenuta 	:= ActualPickingListFromHMI[IdxLista].SupportPianoLegno.ZDim+20;
													WorkAreaState[j].Supporto.DimVertice 			:= ActualPickingListFromHMI[IdxLista].SupportPianoLegno.DimVertice;
													WorkAreaState[j].Supporto.HMAX 					:= ActualPickingListFromHMI[IdxLista].SupportPianoLegno.HMAX;
													WorkAreaState[j].Supporto.Tipologia 			:=  e_Tipo_Pallet.CASSA_STANDARD;//ActualPickingListFromHMI[1].Support.Tipologia;
													WorkAreaState[j].Supporto.XDim 					:= ActualPickingListFromHMI[IdxLista].SupportPianoLegno.XDim;
													WorkAreaState[j].Supporto.YDim 					:= ActualPickingListFromHMI[IdxLista].SupportPianoLegno.YDim;
													WorkAreaState[j].Supporto.ZDim 					:= ActualPickingListFromHMI[IdxLista].SupportPianoLegno.ZDim;
													WorkAreaOffset[j].Y 							:= OFFSET_POSTAZIONE_LEGNO + ActualPickingListFromHMI[IdxLista].SupportPianoLegno.YDim/2;//ATTENZIONE!!! per poter lavorare in centro con i supporti pari, questa misura è la distanza tra il riscontro bundle verticale e il centro postazione PARI
												(* Se ho una cassa pianale in ferro su supporto *)
												TELAIO_PIANO:
													WorkAreaState[j].Supporto.Code 					:= ActualPickingListFromHMI[IdxLista].SupportPianoFerro.Code;
													WorkAreaState[j].Supporto.DimBaseUtile		 	:= ActualPickingListFromHMI[IdxLista].SupportPianoFerro.DimBaseUtile;
													WorkAreaState[j].Supporto.AltezzaDenteRitenuta 	:= ActualPickingListFromHMI[IdxLista].SupportPianoFerro.ZDim+20;
													WorkAreaState[j].Supporto.DimVertice 			:= ActualPickingListFromHMI[IdxLista].SupportPianoFerro.DimVertice;
													WorkAreaState[j].Supporto.HMAX 					:= ActualPickingListFromHMI[IdxLista].SupportPianoFerro.HMAX;
													WorkAreaState[j].Supporto.Tipologia 			:=  e_Tipo_Pallet.CASSA_STANDARD;//ActualPickingListFromHMI[1].Support.Tipologia;
													WorkAreaState[j].Supporto.XDim 					:= ActualPickingListFromHMI[IdxLista].SupportPianoFerro.XDim;
													WorkAreaState[j].Supporto.YDim 					:= ActualPickingListFromHMI[IdxLista].SupportPianoFerro.YDim;
													WorkAreaState[j].Supporto.ZDim 					:= ActualPickingListFromHMI[IdxLista].SupportPianoFerro.ZDim;
													WorkAreaOffset[j].Y 							:= OFFSET_POSTAZIONE_TELAIO - ActualPickingListFromHMI[IdxLista].SupportPianoFerro.YDim/2;//ATTENZIONE!!! per poter lavorare in centro con i supporti pari, questa misura è la distanza tra il riscontro bundle verticale e il centro postazione PARI
												(* Se ho un bundle *)
												BUNDLE_VERT:
													//WorkAreaState[j].P := ElementiDaDepositare;
													WorkAreaState[j].Supporto.Code 					:= ActualPickingListFromHMI[IdxLista].SupportVertBundle.Code;
													WorkAreaState[j].Supporto.DimBaseUtile		 	:= ActualPickingListFromHMI[IdxLista].SupportVertBundle.DimBaseUtile;
													WorkAreaState[j].Supporto.AltezzaDenteRitenuta 	:= ActualPickingListFromHMI[IdxLista].SupportVertBundle.ZDim+20;
													WorkAreaState[j].Supporto.DimVertice 			:= ActualPickingListFromHMI[IdxLista].SupportVertBundle.DimVertice;
													WorkAreaState[j].Supporto.HMAX 					:= ActualPickingListFromHMI[IdxLista].SupportVertBundle.HMAX;
													WorkAreaState[j].Supporto.Tipologia 			:= e_Tipo_Pallet.BUNDLE;//ActualPickingListFromHMI.SupportVert.Tipologia;
													WorkAreaState[j].Supporto.XDim 					:= ActualPickingListFromHMI[IdxLista].SupportVertBundle.XDim;
													WorkAreaState[j].Supporto.YDim 					:= ActualPickingListFromHMI[IdxLista].SupportVertBundle.YDim;
													WorkAreaState[j].Supporto.ZDim 					:= ActualPickingListFromHMI[IdxLista].SupportVertBundle.ZDim;
													WorkAreaState[j].Supporto.ZDim_Ext1        		:= WorkAreaState[j].Supporto.ZDim + 20;	
													//**Lo Que Habia
													WorkAreaOffset[j].Y 							:= 0;
													//Mod 25/&/2025	  
													//WorkAreaOffset[j].Y 		:= ActualPickingListFromHMI[IdxLista].SupportVertBundle.YDim-ActualPickingListFromHMI[IdxLista].SupportVertBundle.DimBaseUtile -40;					
												(* Se ho un A_Frame *)	  
												A_FRAME_VERT:  						
													//WorkAreaState[j].P := ElementiDaDepositare;
													WorkAreaState[j].Supporto.Code 					:= ActualPickingListFromHMI[IdxLista].SupportVertCav.Code;
													WorkAreaState[j].Supporto.DimBaseUtile		 	:= ActualPickingListFromHMI[IdxLista].SupportVertCav.DimBaseUtile;
													WorkAreaState[j].Supporto.AltezzaDenteRitenuta 	:= ActualPickingListFromHMI[IdxLista].SupportVertCav.ZDim+20;
													WorkAreaState[j].Supporto.DimVertice 			:= ActualPickingListFromHMI[IdxLista].SupportVertCav.DimVertice;
													WorkAreaState[j].Supporto.HMAX 					:= ActualPickingListFromHMI[IdxLista].SupportVertCav.HMAX;
													WorkAreaState[j].Supporto.Tipologia 			:= CAVALLETTO;//ActualPickingListFromHMI.SupportVertCav.Tipologia;
													WorkAreaState[j].Supporto.XDim 					:= ActualPickingListFromHMI[IdxLista].SupportVertCav.XDim;
													WorkAreaState[j].Supporto.YDim 					:= ActualPickingListFromHMI[IdxLista].SupportVertCav.YDim;
													WorkAreaState[j].Supporto.ZDim 					:= ActualPickingListFromHMI[IdxLista].SupportVertCav.ZDim;
													WorkAreaState[j].Supporto.ZDim_Ext1        		:= WorkAreaState[j].Supporto.ZDim + 20;	
													WorkAreaState[j].Supporto.TipoTrabajoLado_Cavallete := HMI_WorkAreaDataPicking[j].TipoTrabajoLado_Cavallete ;	
													WorkAreaOffset[j].Y 							:= OFFSET_POSTAZIONE_LEGNO + ActualPickingListFromHMI[IdxLista].SupportVertCav.YDim/2;//ATTENZIONE!!! per poter lavorare in centro con i supporti pari, questa misura è la distanza tra il riscontro bundle verticale e il centro postazione PARI
												   CoordenadaPasillo0_Y := WorkArea[j].Y +  WorkAreaOffset[j].Y  - Dimensioni_Pinza.Spessore - INGOMBRO_RISCONTRO_BUNDLE - WorkAreaState[j].Supporto.YDim /2 ;
													CoordenadaPasillo180_Y := WorkArea[j].Y + WorkAreaState[j].Supporto.YDim /2 + WorkAreaOffset[j].Y  + Dimensioni_Pinza.Spessore + INGOMBRO_RISCONTRO_FRAME  ;	
												
											END_CASE
													  
											WorkAreaProductionList[j].Support := HMI_Formatura.HMI_Forming_Supporto;
										END_IF
									END_IF
									TFClearApprendimento(ADR(WorkAreaState[j].Apprendimento));//Azzeramento apprendimento
								END_FOR
								EXIT; 
						END_CASE // case Pricipal1
					END_IF	//-------->	 //-------> Palet destino
				END_FOR//----------For 1 HMI_WorkAreaDataPicking[i].Destinazione 
				
				Picking.Cmd_CalcolaLista[IdxLista] := TRUE;
				Temp_UDINT[8] := IdxLista;
				HMI_Forming_Attivazione[IdxLista] := TRUE;//attivo nuova formatura
			END_IF //------------------------------ActualPickingListFromHMI[IdxLista].State = e_StatoWorkOrder.DA_ESEGUIRE 
{endregion }



			Temp_UINT[9]	 := 0 ; // añadido
				 
			
			//una volta calcolata la lista per stabilire le postazioni di prelievo e quella di deposito, calcolo la formatura della postazione di deposito
			IF Picking.Cmd_CalcolaLista[IdxLista] THEN
				Temp_UINT[9]	 := IdxLista ;
				Temp_UINT[7] := j ;
				//CASE HMI_WorkAreaDataPicking[NumPostazioneDeposito].Typology OF 	 
				//CASE HMI_WorkAreaDataPicking[j].Typology OF 
				CASE HMI_WorkAreaDataPicking[NumPostazioneDeposito].Typology OF 
					TELAIO_PIANO:
						HMI_Formatura.HMI_Forming_Supporto.Code				:= RequestPickingListFromHMI[IdxLista].SupportPianoFerro.Code;
						HMI_Formatura.HMI_Forming_Supporto.XDim				:= RequestPickingListFromHMI[IdxLista].SupportPianoFerro.XDim;
						HMI_Formatura.HMI_Forming_Supporto.YDim				:= RequestPickingListFromHMI[IdxLista].SupportPianoFerro.YDim;
						HMI_Formatura.HMI_Forming_Supporto.ZDim				:= RequestPickingListFromHMI[IdxLista].SupportPianoFerro.ZDim;
						HMI_Formatura.HMI_Forming_Supporto.DimBaseUtile		:= RequestPickingListFromHMI[IdxLista].SupportPianoFerro.DimBaseUtile;
						HMI_Formatura.HMI_Forming_Supporto.DimVertice 		:= RequestPickingListFromHMI[IdxLista].SupportPianoFerro.DimVertice;
						HMI_Formatura.HMI_Forming_Supporto.HMAX 			:= RequestPickingListFromHMI[IdxLista].SupportPianoFerro.HMAX;
						HMI_Formatura.HMI_Forming_Supporto.Tipologia		:= e_Tipo_Pallet.CASSA_STANDARD;// RequestPickingListFromHMI[1].Support.Tipologia;		

					A_FRAME_VERT:
						HMI_Formatura.HMI_Forming_Supporto.Code				:= RequestPickingListFromHMI[IdxLista].SupportVertCav.Code;
						HMI_Formatura.HMI_Forming_Supporto.XDim				:= RequestPickingListFromHMI[IdxLista].SupportVertCav.XDim;
						HMI_Formatura.HMI_Forming_Supporto.YDim				:= RequestPickingListFromHMI[IdxLista].SupportVertCav.YDim;
						HMI_Formatura.HMI_Forming_Supporto.ZDim				:= RequestPickingListFromHMI[IdxLista].SupportVertCav.ZDim;
						HMI_Formatura.HMI_Forming_Supporto.TipoPianoAppoggio 		:= 1;                      
						HMI_Formatura.HMI_Forming_Supporto.AltezzaDenteRitenuta		:= 15;              
						HMI_Formatura.HMI_Forming_Supporto.ZDim_Ext1        := HMI_Formatura.HMI_Forming_Supporto.ZDim + HMI_Formatura.HMI_Forming_Supporto.AltezzaDenteRitenuta;
						HMI_Formatura.HMI_Forming_Supporto.DimBaseUtile		:= RequestPickingListFromHMI[IdxLista].SupportVertCav.DimBaseUtile;
						HMI_Formatura.HMI_Forming_Supporto.DimVertice 		:= RequestPickingListFromHMI[IdxLista].SupportVertCav.DimVertice;
						HMI_Formatura.HMI_Forming_Supporto.HMAX 			:= RequestPickingListFromHMI[IdxLista].SupportVertCav.HMAX;
						HMI_Formatura.HMI_Forming_Supporto.Tipologia 		:= e_Tipo_Pallet.CAVALLETTO;                  
			
					BUNDLE_VERT:
						HMI_Formatura.HMI_Forming_Supporto.Code				:= RequestPickingListFromHMI[IdxLista].SupportVertBundle.Code;
						HMI_Formatura.HMI_Forming_Supporto.XDim				:= RequestPickingListFromHMI[IdxLista].SupportVertBundle.XDim;
						HMI_Formatura.HMI_Forming_Supporto.YDim				:= RequestPickingListFromHMI[IdxLista].SupportVertBundle.YDim*2;
						HMI_Formatura.HMI_Forming_Supporto.ZDim				:= RequestPickingListFromHMI[IdxLista].SupportVertBundle.ZDim;
						HMI_Formatura.HMI_Forming_Supporto.TipoPianoAppoggio := 1;                      
						HMI_Formatura.HMI_Forming_Supporto.AltezzaDenteRitenuta		:= 20;              
						HMI_Formatura.HMI_Forming_Supporto.ZDim_Ext1        := HMI_Formatura.HMI_Forming_Supporto.ZDim +	HMI_Formatura.HMI_Forming_Supporto.AltezzaDenteRitenuta;
						HMI_Formatura.HMI_Forming_Supporto.DimBaseUtile		:= RequestPickingListFromHMI[IdxLista].SupportVertBundle.DimBaseUtile;
						HMI_Formatura.HMI_Forming_Supporto.DimVertice 		:= RequestPickingListFromHMI[IdxLista].SupportVertBundle.DimVertice*2;
						HMI_Formatura.HMI_Forming_Supporto.HMAX 			:= RequestPickingListFromHMI[IdxLista].SupportVertBundle.HMAX;
						HMI_Formatura.HMI_Forming_Supporto.Tipologia 		:= e_Tipo_Pallet.BUNDLE;                  
						HMI_Formatura.HMI_Forming_Supporto.LatoDeposito 	:= 180;                     
					ELSE	
						HMI_Formatura.HMI_Forming_Supporto.Code				:= RequestPickingListFromHMI[IdxLista].SupportPianoLegno.Code;
						HMI_Formatura.HMI_Forming_Supporto.XDim				:= RequestPickingListFromHMI[IdxLista].SupportPianoLegno.XDim;
						HMI_Formatura.HMI_Forming_Supporto.YDim				:= RequestPickingListFromHMI[IdxLista].SupportPianoLegno.YDim;
						HMI_Formatura.HMI_Forming_Supporto.ZDim				:= RequestPickingListFromHMI[IdxLista].SupportPianoLegno.ZDim;
						HMI_Formatura.HMI_Forming_Supporto.DimBaseUtile		:= RequestPickingListFromHMI[IdxLista].SupportPianoLegno.DimBaseUtile;
						HMI_Formatura.HMI_Forming_Supporto.DimVertice 		:= RequestPickingListFromHMI[IdxLista].SupportPianoLegno.DimVertice;
						HMI_Formatura.HMI_Forming_Supporto.HMAX 			:= RequestPickingListFromHMI[IdxLista].SupportPianoLegno.HMAX;
						HMI_Formatura.HMI_Forming_Supporto.Tipologia		:= e_Tipo_Pallet.CASSA_STANDARD;// RequestPickingListFromHMI[1].Support.Tipologia;		
				END_CASE	
				WorkAreaProductionList[j].Support := HMI_Formatura.HMI_Forming_Supporto;		   
				//WorkAreaProductionList[NumPostazioneDeposito].Support := HMI_Formatura.HMI_Forming_Supporto;												 
				//
				HMI_Formatura.HMI_Forming_LastraDaDepositare.XDim		:= RequestPickingListFromHMI[IdxLista].SlabDimension.XDim;
				HMI_Formatura.HMI_Forming_LastraDaDepositare.YDim		:= RequestPickingListFromHMI[IdxLista].SlabDimension.YDim;
				HMI_Formatura.HMI_Forming_LastraDaDepositare.ZDim		:= RequestPickingListFromHMI[IdxLista].SlabDimension.ZDim;
																									
				HMI_Formatura.HMI_Forming_CodiciAbilitatiFormatura[IdxLista].Code[1] := 1;                 
				
				FaldaDaDepositare.TypologyCode := RequestPickingListFromHMI[IdxLista].Layer.Tipologia;
				
				FaldaDaDepositare.XDim := RequestPickingListFromHMI[IdxLista].Layer.XDim;
				FaldaDaDepositare.YDim := RequestPickingListFromHMI[IdxLista].Layer.YDim;
				FaldaDaDepositare.ZDim := RequestPickingListFromHMI[IdxLista].Layer.ZDim;
				
				//Vado ad assegnare il numero giusto di elementi a seconda se è presente o meno la falda 
				IF (RequestPickingListFromHMI[IdxLista].LayerSequence = 1 AND HMI_AbilitaDepositoFalda) AND RequestPickingListFromHMI[IdxLista].SupportPianoLegno.Tipologia <> CAVALLETTO AND RequestPickingListFromHMI[IdxLista].SupportPianoLegno.Tipologia <> BUNDLE THEN 
					HMI_Formatura.HMI_Forming_NumeroElementiDaDepositare	:= TO_UINT(2*RequestPickingListFromHMI[IdxLista].SlabNumber - 1);
				ELSE 
					HMI_Formatura.HMI_Forming_NumeroElementiDaDepositare	:= TO_UINT(RequestPickingListFromHMI[IdxLista].SlabNumber);
				END_IF
				
				//Ack 
				IF HMI_ErrAckCalcolaFormatura THEN
					HMI_Forming_ErroreCalcoli := 0;
					HMI_ErrAckCalcolaFormatura := FALSE;
					FOR i:= 1 TO MAXFORMING DO
						HMI_ConfermaAttivazioneFormatura[i] := FALSE;
						HMI_Forming_FormaturaAttivata[i] := FALSE;
					END_FOR
				END_IF
				
				//Azzeramento comandi in caso di errore
				IF HMI_Forming_ErroreCalcoli <> 0 THEN
					FOR i:=1 TO MAXFORMING DO
						HMI_Forming_Attivazione[i] 		:= FALSE;
						HMI_Forming_Disattivazione[i] 	:= FALSE;
					END_FOR
					HMI_Forming_Calcola 			:= FALSE;
				END_IF
				
				//Valorizzo altezza esterna supporto
				//IF HMI_Forming_Supporto.ZDim_Ext1 = 0 THEN
					HMI_Forming_Supporto.ZDim_Ext1 := HMI_Forming_Supporto.ZDim + HMI_Forming_Supporto.AltezzaDenteRitenuta;
				//END_IF
				//Valorizzo HMAX x tipologia pallet
				IF HMI_Forming_Supporto.Tipologia = PALLET_STANDARD THEN
					HMI_Forming_Supporto.HMAX := HMI_Forming_Supporto.ZDim;
				END_IF

				
//##########################################################################################		  
//------------------------------------------------------------------------------------------				
///////////	Attivazione	Formature  autosettata dopo caricamento dei dati dell'ordine  /////
//------------------------------------------------------------------------------------------	
					 
				//FOR i:= 1 TO MAXFORMING DO
					idxForm:= IdxLista;//forzo a 1 la formatura da attivare
					IF HMI_Forming_Attivazione[idxForm] AND idxForm <=3 AND NOT Formacion_De_listaOk[idxForm] THEN
						Forming[idxForm] := FormingEmpty;
						(*IF NOT CalcolaFormaturaTrig AND TFCalcoloFormaturaDaLista.PulisciMemoriaDone THEN *)//#Modificado
							 IF TFCalcoloFormaturaDaLista.CalcolaFormaturaDone THEN
								CalcolaFormaturaTrig := TRUE;	  
							END_IF	
						IF NOT CalcolaFormaturaTrig  AND NOT Formacion_De_listaOk[idxForm] THEN 
							HMI_Forming_FormaturaAttivata[idxForm] 	:= FALSE;
							TFCalcoloFormaturaDaLista.PulisciMemoria 	:= TRUE;
							IF TFCalcoloFormaturaDaLista.PulisciMemoriaDone THEN	
								HMI_Forming_ErroreCalcoli := 0;
								CalcolaFormaturaTrig := TRUE;
								IF (RequestPickingListFromHMI[1].LayerSequence = 0 OR NOT HMI_AbilitaDepositoFalda)
									AND HMI_Forming_NumeroElementiDaDepositare >0 
								THEN
									//Assegno l'ordine tutto a 1 perchè ho solo lastre	
									FOR i:= 1 TO MAXFORMINGSLAB DO
										//IF i <= HMI_Forming_NumeroElementiDaDepositare THEN
										IF i <= HMI_Forming_NumeroElementiDaDepositare + HMI_NumeroPezziPresentiPostazione[NumPostazioneDeposito] THEN
										//IF i <= 20THEN
											TFCalcoloFormaturaDaLista.TipoElementoDep[i] := LASTRA;//Settiamo tutte lastre!!
										ELSE
											TFCalcoloFormaturaDaLista.TipoElementoDep[i] := TERMINATORE;//Settiamo il resto come terminatore
										END_IF
									END_FOR
								ELSE
									//FOR i := 1 TO HMI_Forming_NumeroElementiDaDepositare DO//BY (Request_WorkOrder.LayerSequence+1) DO		  
									FOR i := 1 TO HMI_Forming_NumeroElementiDaDepositare DO//BY (Request_WorkOrder.LayerSequence+1) DO
										IF i MOD 2 = 1 THEN// i <= HMI_Forming_NumeroElementiDaDepositare THEN 
											TFCalcoloFormaturaDaLista.TipoElementoDep[i] := LASTRA;//Settiamo tipo lastre!!
										ELSE
											TFCalcoloFormaturaDaLista.TipoElementoDep[i] := FALDA;//Settiamo tipoi falda!
										END_IF
										TFCalcoloFormaturaDaLista.TipoElementoDep[i+1] := TERMINATORE;//Settiamo il resto come terminatore
									END_FOR
								END_IF	
								//FOR i := HMI_Forming_NumeroElementiDaDepositare+1 TO MAXFORMINGSLAB DO
								FOR i := (HMI_Forming_NumeroElementiDaDepositare + HMI_NumeroPezziPresentiPostazione[NumPostazioneDeposito] )   +1 TO MAXFORMINGSLAB DO
									TFCalcoloFormaturaDaLista.TipoElementoDep[i] := TERMINATORE;//Settiamo il resto come terminatore
								END_FOR
									
								TFCalcoloFormaturaDaLista.Materiale[e_Tipo_Elemento_Da_Lavorare.LASTRA]		:= HMI_Forming_LastraDaDepositare; 
								TFCalcoloFormaturaDaLista.Materiale[e_Tipo_Elemento_Da_Lavorare.FALDA]		:= FaldaDaDepositare;
								TFCalcoloFormaturaDaLista.Materiale[e_Tipo_Elemento_Da_Lavorare.QUADROTTA]	:= HMI_Forming_LastraDaDepositare;
								TFCalcoloFormaturaDaLista.Supporto											:= HMI_Forming_Supporto;	//Assegno la tipologia di supporto
								
								//CASE HMI_WorkAreaDataPicking[j].Typology OF //**Mod	 
								CASE HMI_WorkAreaDataPicking[NumPostazioneDeposito].Typology OF //**Mod
									BUNDLE_VERT:
										TFCalcoloFormaturaDaLista.TipoOrdinamento := 4;//Ordinamento di deposito òato 180°
									A_FRAME_VERT:
										TFCalcoloFormaturaDaLista.TipoOrdinamento := 1;//Ordinamento di deposito, prima un lato poi l'altro	
										TFCalcoloFormaturaDaLista.HabiCalTodasCordenadas := TRUE ;
									ELSE
										TFCalcoloFormaturaDaLista.TipoOrdinamento := 2;//Ordinamento di deposito consecutivo	 
								END_CASE
									 
								TFCalcoloFormaturaDaLista.CalcolaFormatura := TRUE; 		//Lancio esecuzione dei calcoli
								MEMSET(ADR(HMI_Forming_FormaturaCalcolata),0,SIZEOF(HMI_Forming_FormaturaCalcolata));	//Pulisco la memoria di destinazione
								HMI_Forming_Attivazione[i] := FALSE;
								TFCalcoloFormaturaDaLista.PulisciMemoria := FALSE;
							END_IF
						ELSIF (TFCalcoloFormaturaDaLista.CalcolaFormaturaDone OR TFCalcoloFormaturaDaLista.Errore > 0) AND CalcolaFormaturaTrig AND NOT Formacion_De_listaOk[idxForm] THEN
							CalcolaFormaturaTrig := FALSE;
							TFCalcoloFormaturaDaLista.CalcolaFormatura := FALSE;
							Formacion_De_listaOk[idxForm] := TRUE ;
							IF TFCalcoloFormaturaDaLista.Errore = 0 THEN
								IDFormatura 								:= IDFormatura+1;
								GUIDFormatura 								:= STRING_TO_UINT(concat(UINT_TO_STRING(NUMERO_MACCHINA),UINT_TO_STRING(IDFormatura)));
								HMI_Forming_GUID 							:= GUIDFormatura;
						
								HMI_Forming_FormaturaCalcolata 				:= TFCalcoloFormaturaDaLista.FormingSlab;
								Forming[idxForm] 							:= FormingEmpty;	//Pulisco la memoria di destinazione
								Forming[idxForm] 							:= TFCalcoloFormaturaDaLista.FormingSlab;
								Forming[idxForm].Enable 					:= 1;
								Forming[idxForm].Code 						:= HMI_Forming_CodiciAbilitatiFormatura[idxForm].Code;
								Forming[idxForm].GUID						:= HMI_Forming_GUID;
								Forming[idxForm].Pallet						:= HMI_Forming_Supporto;
								HMI_Forming_IndiceFormaturaAttivata := idxForm;
								HMI_Forming_FormaturaAttivata[idxForm] 	:= TRUE;
								HMI_ConfermaAttivazioneFormatura[idxForm] := TRUE;
								//Valorizzo la struttura del WAPL per ogni elemento da elaborare
								FOR jj := 1 TO MAXELEMENTLIST DO
									IF jj < ElementiElaborati[IdxLista] THEN
										WorkAreaProductionList[NumPostazioneDeposito].PElementList[jj].PElement 		:= TFCalcoloFormaturaDaLista.FormingSlab.PElement[jj];	
										WorkAreaProductionList[NumPostazioneDeposito].PElementList[jj].Stato			:= ELEMENTO_DA_ELABORARE;
									
										IF Picking.HMI_PareggiaturaLastraAbilitata THEN
											WorkAreaProductionList[NumPostazioneDeposito].PElementList[jj].Pareggiatura := PAREGGIATURA_DA_ESEGUIRE;
										ELSE
											WorkAreaProductionList[NumPostazioneDeposito].PElementList[jj].Pareggiatura := PAREGGIATURA_DISABILITATA;
										END_IF
									ELSE
										WorkAreaProductionList[NumPostazioneDeposito].PElementList[jj].Stato			:= ELEMENTO_NOT_DEFINED;
									END_IF
								END_FOR
							ELSE
								HMI_Forming_ErroreCalcoli := TFCalcoloFormaturaDaLista.Errore;
							END_IF
							HMI_Forming_Attivazione[idxForm] := FALSE;
						END_IF
					ELSIF HMI_Forming_Attivazione[idxForm]  AND NOT Formacion_De_listaOk[idxForm] THEN
						memset(destAddr:=ADR(TFCalcoloFormaturaDaLista.Errore),fillByte:=(UINT_TO_USINT(ErrNumeroMassimoFormatureAmmesse)),n:=SIZEOF(TFCalcoloFormaturaDaLista.Errore));
					END_IF
				
					//Disattivazione formatura
					IF HMI_Forming_Disattivazione[idxForm] THEN
						HMI_Forming_Disattivazione[idxForm] := FALSE;
						Forming[idxForm] := FormingEmpty;	//Pulisco la formatura selezionata e di consegenza la disattivo
					END_IF
						
				//END_FOR
				
//####################################################################						 

						  
				(* Metto in stato di esecuzione il nuovo W.O. se tutto si è attivato *)
				IF HMI_Forming_FormaturaAttivata[IdxLista] THEN

					ActualPickingListFromHMI[IdxLista].State := e_StatoWorkOrder.DA_ESEGUIRE;
					//Azzero le liste per le postazioni dove non avviene la pallettizzazione
					FOR i:= Iforstart TO Iforend DO		 
						WorkAreaProductionList[i].Stato := e_Stato_ListaDiProduzione.LISTA_PROD_ASSENTE;
					END_FOR
					//WorkAreaProductionList[NumPostazioneDeposito].Support := Forming[idxForm].Pallet;
					WorkAreaProductionList[NumPostazioneDeposito].Stato 					:= LISTA_PROD_DA_ESEGUIRE;
					WorkAreaProductionList[NumPostazioneDeposito].NumeroListaAssociata 		:= IdxLista;
					WorkAreaState[NumPostazioneDeposito].F 									:= idxForm;
					Picking.Cmd_CalcolaLista[IdxLista] 										:= FALSE;
					HMI_Forming_FormaturaAttivata[IdxLista] 								:= FALSE;
					//CalcolaFormingRT[IdxLista] 												:= TRUE;
				END_IF
				//TFCalcoloFormaturaDaLista();
			END_IF	
		
			TFCalcoloFormaturaDaLista();
		END_IF	
		
		//verifico che la lista sia in esecuzione o terminata
		IF NOT ListaInEsecuzione[IdxLista] THEN
			FOR i:= Iforstart TO Iforend DO	
				IF WorkAreaProductionList[i].Stato = e_Stato_ListaDiProduzione.LISTA_PROD_IN_ESECUZIONE THEN
					ListaInEsecuzione[IdxLista] := TRUE;
					EXIT;	
				END_IF
			END_FOR
		ELSE
			FOR i:= Iforstart TO Iforend DO	
				IF WorkAreaProductionList[i].Stato = e_Stato_ListaDiProduzione.LISTA_PROD_ESEGUITA THEN
					ListaInEsecuzione[IdxLista] := FALSE;
					EXIT;	
				END_IF
			END_FOR
		END_IF
		
		//
		FOR i:= Iforstart TO Iforend DO	
			IF NumeroPezziPresentiPostazioneStart[i] = 0 AND WorkAreaState[i].P > 1 THEN
				NumeroPezziPresentiPostazioneStart[i] := TO_UINT(WorkAreaState[i].P);
			END_IF
		
			IF NOT HMI_WorkAreaDataPicking[i].Destinazione THEN
				IF HMI_WorkAreaDataPicking[i].NumElementiDaLavorare > 0 THEN
					//IF HMI_WorkAreaDataPicking[i].NumElementiDaLavorare >= TO_UINT(WorkAreaState[i].P)-1 THEN
					//	HMI_NumeroLastreRimanentiOrdineAttuale[i] := HMI_WorkAreaDataPicking[i].NumElementiDaLavorare - TO_UINT(WorkAreaState[i].P);
					//ELSE
					//	HMI_NumeroLastreRimanentiOrdineAttuale[i] := 0;
					//END_IF
					IF HMI_WorkAreaDataPicking[i].NumElementiDaLavorare - (TO_UINT(WorkAreaState[i].P) - NumeroPezziPresentiPostazioneStart[i]) > 0 THEN
						HMI_NumeroLastreRimanentiOrdineAttuale[i] := MIN(HMI_WorkAreaDataPicking[i].NumElementiDaLavorare,HMI_WorkAreaDataPicking[i].NumElementiDaLavorare - 
																	(NumeroPezziPresentiPostazioneStart[i] - TO_UINT(WorkAreaState[i].P)));
					ELSE
						HMI_NumeroLastreRimanentiOrdineAttuale[i] := 0;
					END_IF
				ELSE
					HMI_NumeroLastreRimanentiOrdineAttuale[i] := 0;
				END_IF
			ELSE
				IF NumeroPezziPresentiPostazioneStart[i] <= (TO_UINT(WorkAreaState[i].P)) AND NumeroPezziPresentiPostazioneStart[i]>0 THEN
					HMI_NumeroLastreRimanentiOrdineAttuale[i] := TO_UINT(WorkAreaState[i].P) - NumeroPezziPresentiPostazioneStart[i]+1;
				ELSE
					HMI_NumeroLastreRimanentiOrdineAttuale[i] := 0;
				END_IF
			END_IF
			IF (WorkAreaProductionList[i].Stato = e_Stato_ListaDiProduzione.LISTA_PROD_IN_ESECUZIONE OR WorkAreaProductionList[i].Stato = e_Stato_ListaDiProduzione.LISTA_PROD_ESEGUITA) AND WorkAreaState[i].P > 1 THEN
					//P:	(* Pack Pointer - Puntatore tabella ELEMENTO (0..n-1=, -1 dato non valido),Numero ELEMENTO successivo da depositare *)
					HMI_NumeroLastreDepOrdineAttuale[IdxLista] := TO_UINT(WorkAreaState[i].P-1);
				IF NumeroPezziPresentiPostazioneStart[i] < (TO_UINT(WorkAreaState[i].P)) AND NumeroPezziPresentiPostazioneStart[i]>0 THEN
					HMI_NumeroLastreDepOrdineAttuale[IdxLista] := TO_UINT(WorkAreaState[i].P) - NumeroPezziPresentiPostazioneStart[i];
				ELSE
					HMI_NumeroLastreDepOrdineAttuale[IdxLista] := TO_UINT(WorkAreaState[i].P) - 1;
				END_IF
			END_IF	
		END_FOR
		
		//trasferisco i valori alla variabile in lettura x HMI
		MEMCPY(destAddr:=ADR(HMI_WorkAreaProductionList),srcAddr:=ADR(WorkAreaProductionList),n:=SIZEOF(HMI_WorkAreaProductionList));
		//IF CalcolaFormingRT[IdxLista] AND NOT CalcolaFormingRT2[IdxLista] THEN //original	
			 
				  
					   
		//##################################añadido	############################################################ 
		IF 	NOT CalcolaFormingRT[IdxLista] AND NOT CalcolaFormingRT2[IdxLista] AND Temp_UINT[9] = IdxLista THEN
			
				CalcolaFormaturaTrig2 		:= FALSE ;
				CalcolaFormingRT[IdxLista] 	:= TRUE ;
	 
		END_IF
  		//#######################################################################################################
					   
							
